LIN {X 27.783,Y -37.308,Z -57.523,A -90.000,B 90.000,C 0.000} C_DIS
LIN {X 27.828,Y -37.308,Z -57.428,A -90.000,B 90.000,C 0.000} C_DIS
LIN {X 28.026,Y -37.308,Z -57.054,A -90.000,B 90.000,C 0.000} C_DIS
LIN {X 28.266,Y -37.308,Z -56.705,A -90.000,B 90.000,C 0.000} C_DIS
LIN {X 28.546,Y -37.308,Z -56.387,A -90.000,B 90.000,C 0.000} C_DIS
LIN {X 28.652,Y -37.308,Z -56.277,A -90.000,B 90.000,C 0.000} C_DIS
LIN {X 28.954,Y -37.308,Z -56.010,A -90.000,B 90.000,C 0.000} C_DIS
LIN {X 29.286,Y -37.308,Z -55.783,A -90.000,B 90.000,C 0.000} C_DIS
LIN {X 29.386,Y -37.308,Z -55.729,A -90.000,B 90.000,C 0.000} C_DIS
LIN {X 29.854,Y -37.308,Z -55.488,A -90.000,B 90.000,C 0.000} C_DIS
LIN {X 30.232,Y -37.308,Z -55.349,A -90.000,B 90.000,C 0.000} C_DIS
LIN {X 30.624,Y -37.308,Z -55.258,A -90.000,B 90.000,C 0.000} C_DIS
LIN {X 30.794,Y -37.308,Z -55.228,A -90.000,B 90.000,C 0.000} C_DIS
LIN {X 30.962,Y -37.308,Z -55.200,A -90.000,B 90.000,C 0.000} C_DIS
LIN {X 31.362,Y -37.308,Z -55.158,A -90.000,B 90.000,C 0.000} C_DIS
LIN {X 31.411,Y -37.308,Z -55.158,A -90.000,B 90.000,C 0.000} C_DIS
LIN {X 31.494,Y -37.308,Z -54.811,A -90.000,B 90.000,C 0.000} C_DIS
LIN {X 31.553,Y -37.308,Z -54.530,A -90.000,B 90.000,C 0.000} C_DIS
LIN {X 31.658,Y -37.308,Z -54.086,A -90.000,B 90.000,C 0.000} C_DIS
LIN {X 31.702,Y -37.308,Z -53.930,A -90.000,B 90.000,C 0.000} C_DIS
LIN {X 31.754,Y -37.308,Z -53.727,A -90.000,B 90.000,C 0.000} C_DIS
LIN {X 31.943,Y -37.308,Z -53.228,A -90.000,B 90.000,C 0.000} C_DIS
LIN {X 32.172,Y -37.308,Z -52.712,A -90.000,B 90.000,C 0.000} C_DIS
LIN {X 32.257,Y -37.308,Z -52.537,A -90.000,B 90.000,C 0.000} C_DIS
LIN {X 32.455,Y -37.308,Z -52.163,A -90.000,B 90.000,C 0.000} C_DIS
LIN {X 32.688,Y -37.308,Z -51.810,A -90.000,B 90.000,C 0.000} C_DIS
LIN {X 32.928,Y -37.308,Z -51.461,A -90.000,B 90.000,C 0.000} C_DIS
LIN {X 33.080,Y -37.308,Z -51.265,A -90.000,B 90.000,C 0.000} C_DIS
LIN {X 33.360,Y -37.308,Z -50.947,A -90.000,B 90.000,C 0.000} C_DIS
LIN {X 33.675,Y -37.308,Z -50.664,A -90.000,B 90.000,C 0.000} C_DIS
LIN {X 33.699,Y -37.308,Z -50.645,A -90.000,B 90.000,C 0.000} C_DIS
LIN {X 33.882,Y -37.308,Z -50.469,A -90.000,B 90.000,C 0.000} C_DIS
LIN {X 34.204,Y -37.308,Z -50.181,A -90.000,B 90.000,C 0.000} C_DIS
LIN {X 34.543,Y -37.308,Z -49.942,A -90.000,B 90.000,C 0.000} C_DIS
LIN {X 34.924,Y -37.308,Z -49.737,A -90.000,B 90.000,C 0.000} C_DIS
LIN {X 35.239,Y -37.308,Z -49.567,A -90.000,B 90.000,C 0.000} C_DIS
LIN {X 35.593,Y -37.308,Z -49.385,A -90.000,B 90.000,C 0.000} C_DIS
LIN {X 35.987,Y -37.308,Z -49.230,A -90.000,B 90.000,C 0.000} C_DIS
LIN {X 36.396,Y -37.308,Z -49.121,A -90.000,B 90.000,C 0.000} C_DIS
LIN {X 36.614,Y -37.308,Z -49.080,A -90.000,B 90.000,C 0.000} C_DIS
LIN {X 37.252,Y -37.308,Z -48.939,A -90.000,B 90.000,C 0.000} C_DIS
LIN {X 37.671,Y -37.308,Z -48.880,A -90.000,B 90.000,C 0.000} C_DIS
LIN {X 38.095,Y -37.308,Z -48.870,A -90.000,B 90.000,C 0.000} C_DIS
LIN {X 38.607,Y -37.308,Z -48.891,A -90.000,B 90.000,C 0.000} C_DIS
LIN {X 39.150,Y -37.308,Z -48.910,A -90.000,B 90.000,C 0.000} C_DIS
LIN {X 39.644,Y -37.308,Z -48.933,A -90.000,B 90.000,C 0.000} C_DIS
LIN {X 40.080,Y -37.308,Z -49.001,A -90.000,B 90.000,C 0.000} C_DIS
LIN {X 40.577,Y -37.308,Z -49.119,A -90.000,B 90.000,C 0.000} C_DIS
LIN {X 41.623,Y -37.308,Z -49.377,A -90.000,B 90.000,C 0.000} C_DIS
LIN {X 41.811,Y -37.308,Z -49.428,A -90.000,B 90.000,C 0.000} C_DIS
LIN {X 42.485,Y -37.308,Z -49.639,A -90.000,B 90.000,C 0.000} C_DIS
LIN {X 43.044,Y -37.308,Z -49.852,A -90.000,B 90.000,C 0.000} C_DIS
LIN {X 43.197,Y -37.308,Z -49.901,A -90.000,B 90.000,C 0.000} C_DIS
LIN {X 44.006,Y -37.308,Z -50.170,A -90.000,B 90.000,C 0.000} C_DIS
LIN {X 44.597,Y -37.308,Z -50.272,A -90.000,B 90.000,C 0.000} C_DIS
LIN {X 45.346,Y -37.308,Z -50.195,A -90.000,B 90.000,C 0.000} C_DIS
LIN {X 45.719,Y -37.308,Z -50.136,A -90.000,B 90.000,C 0.000} C_DIS
LIN {X 46.852,Y -37.308,Z -49.935,A -90.000,B 90.000,C 0.000} C_DIS
LIN {X 47.253,Y -37.308,Z -49.893,A -90.000,B 90.000,C 0.000} C_DIS
LIN {X 47.873,Y -37.308,Z -49.867,A -90.000,B 90.000,C 0.000} C_DIS
LIN {X 49.033,Y -37.308,Z -49.780,A -90.000,B 90.000,C 0.000} C_DIS
LIN {X 49.435,Y -37.308,Z -49.789,A -90.000,B 90.000,C 0.000} C_DIS
LIN {X 49.834,Y -37.308,Z -49.846,A -90.000,B 90.000,C 0.000} C_DIS
LIN {X 50.766,Y -37.308,Z -50.075,A -90.000,B 90.000,C 0.000} C_DIS
LIN {X 52.001,Y -37.308,Z -50.317,A -90.000,B 90.000,C 0.000} C_DIS
LIN {X 52.390,Y -37.308,Z -50.424,A -90.000,B 90.000,C 0.000} C_DIS
LIN {X 52.762,Y -37.308,Z -50.578,A -90.000,B 90.000,C 0.000} C_DIS
LIN {X 53.137,Y -37.308,Z -50.764,A -90.000,B 90.000,C 0.000} C_DIS
LIN {X 53.494,Y -37.308,Z -50.992,A -90.000,B 90.000,C 0.000} C_DIS
LIN {X 55.027,Y -37.308,Z -51.985,A -90.000,B 90.000,C 0.000} C_DIS
LIN {X 55.470,Y -37.308,Z -52.261,A -90.000,B 90.000,C 0.000} C_DIS
LIN {X 55.828,Y -37.308,Z -52.489,A -90.000,B 90.000,C 0.000} C_DIS
LIN {X 56.155,Y -37.308,Z -52.757,A -90.000,B 90.000,C 0.000} C_DIS
LIN {X 58.129,Y -37.308,Z -54.502,A -90.000,B 90.000,C 0.000} C_DIS
LIN {X 58.427,Y -37.308,Z -54.756,A -90.000,B 90.000,C 0.000} C_DIS
LIN {X 59.623,Y -37.308,Z -55.989,A -90.000,B 90.000,C 0.000} C_DIS
LIN {X 60.678,Y -37.308,Z -57.127,A -90.000,B 90.000,C 0.000} C_DIS
LIN {X 60.841,Y -37.308,Z -57.318,A -90.000,B 90.000,C 0.000} C_DIS
LIN {X 61.095,Y -37.308,Z -57.631,A -90.000,B 90.000,C 0.000} C_DIS
LIN {X 62.907,Y -37.308,Z -59.964,A -90.000,B 90.000,C 0.000} C_DIS
LIN {X 64.082,Y -37.308,Z -61.532,A -90.000,B 90.000,C 0.000} C_DIS
LIN {X 64.569,Y -37.308,Z -62.202,A -90.000,B 90.000,C 0.000} C_DIS
LIN {X 64.776,Y -37.308,Z -62.508,A -90.000,B 90.000,C 0.000} C_DIS
LIN {X 64.823,Y -37.308,Z -62.584,A -90.000,B 90.000,C 0.000} C_DIS
LIN {X 66.473,Y -37.308,Z -65.119,A -90.000,B 90.000,C 0.000} C_DIS
LIN {X 68.094,Y -37.308,Z -67.394,A -90.000,B 90.000,C 0.000} C_DIS
LIN {X 68.483,Y -37.308,Z -67.868,A -90.000,B 90.000,C 0.000} C_DIS
LIN {X 69.055,Y -37.308,Z -68.557,A -90.000,B 90.000,C 0.000} C_DIS
LIN {X 71.014,Y -37.308,Z -70.453,A -90.000,B 90.000,C 0.000} C_DIS
LIN {X 71.187,Y -37.308,Z -70.608,A -90.000,B 90.000,C 0.000} C_DIS
LIN {X 72.017,Y -37.308,Z -71.360,A -90.000,B 90.000,C 0.000} C_DIS
LIN {X 72.363,Y -37.308,Z -71.676,A -90.000,B 90.000,C 0.000} C_DIS
LIN {X 72.612,Y -37.308,Z -71.901,A -90.000,B 90.000,C 0.000} C_DIS
LIN {X 73.661,Y -37.308,Z -72.861,A -90.000,B 90.000,C 0.000} C_DIS
LIN {X 73.970,Y -37.308,Z -73.159,A -90.000,B 90.000,C 0.000} C_DIS
LIN {X 74.840,Y -37.308,Z -74.023,A -90.000,B 90.000,C 0.000} C_DIS
LIN {X 75.190,Y -37.308,Z -74.381,A -90.000,B 90.000,C 0.000} C_DIS
LIN {X 76.260,Y -37.308,Z -75.552,A -90.000,B 90.000,C 0.000} C_DIS
LIN {X 76.316,Y -37.308,Z -75.610,A -90.000,B 90.000,C 0.000} C_DIS
LIN {X 76.816,Y -37.308,Z -76.175,A -90.000,B 90.000,C 0.000} C_DIS
LIN {X 77.048,Y -37.308,Z -76.388,A -90.000,B 90.000,C 0.000} C_DIS
LIN {X 77.183,Y -37.308,Z -76.518,A -90.000,B 90.000,C 0.000} C_DIS
LIN {X 77.358,Y -37.308,Z -76.656,A -90.000,B 90.000,C 0.000} C_DIS
LIN {X 77.467,Y -37.308,Z -76.752,A -90.000,B 90.000,C 0.000} C_DIS
LIN {X 77.895,Y -37.308,Z -76.631,A -90.000,B 90.000,C 0.000} C_DIS
LIN {X 77.919,Y -37.308,Z -76.212,A -90.000,B 90.000,C 0.000} C_DIS
LIN {X 77.968,Y -37.308,Z -75.699,A -90.000,B 90.000,C 0.000} C_DIS
LIN {X 78.002,Y -37.308,Z -75.376,A -90.000,B 90.000,C 0.000} C_DIS
LIN {X 78.021,Y -37.308,Z -75.002,A -90.000,B 90.000,C 0.000} C_DIS
LIN {X 78.090,Y -37.308,Z -74.174,A -90.000,B 90.000,C 0.000} C_DIS
LIN {X 78.188,Y -37.308,Z -73.133,A -90.000,B 90.000,C 0.000} C_DIS
LIN {X 78.240,Y -37.308,Z -72.633,A -90.000,B 90.000,C 0.000} C_DIS
LIN {X 78.304,Y -37.308,Z -72.102,A -90.000,B 90.000,C 0.000} C_DIS
LIN {X 78.457,Y -37.308,Z -71.210,A -90.000,B 90.000,C 0.000} C_DIS
LIN {X 78.569,Y -37.308,Z -70.697,A -90.000,B 90.000,C 0.000} C_DIS
LIN {X 78.787,Y -37.308,Z -69.967,A -90.000,B 90.000,C 0.000} C_DIS
LIN {X 79.031,Y -37.308,Z -69.231,A -90.000,B 90.000,C 0.000} C_DIS
LIN {X 79.184,Y -37.308,Z -68.786,A -90.000,B 90.000,C 0.000} C_DIS
LIN {X 79.235,Y -37.308,Z -68.654,A -90.000,B 90.000,C 0.000} C_DIS
LIN {X 79.791,Y -37.308,Z -67.259,A -90.000,B 90.000,C 0.000} C_DIS
LIN {X 80.485,Y -37.308,Z -65.685,A -90.000,B 90.000,C 0.000} C_DIS
LIN {X 80.643,Y -37.308,Z -65.338,A -90.000,B 90.000,C 0.000} C_DIS
LIN {X 81.438,Y -37.308,Z -63.804,A -90.000,B 90.000,C 0.000} C_DIS
LIN {X 81.684,Y -37.308,Z -63.383,A -90.000,B 90.000,C 0.000} C_DIS
LIN {X 82.705,Y -37.308,Z -61.742,A -90.000,B 90.000,C 0.000} C_DIS
LIN {X 84.243,Y -37.308,Z -59.630,A -90.000,B 90.000,C 0.000} C_DIS
LIN {X 85.732,Y -37.308,Z -57.856,A -90.000,B 90.000,C 0.000} C_DIS
LIN {X 86.059,Y -37.308,Z -57.494,A -90.000,B 90.000,C 0.000} C_DIS
LIN {X 87.795,Y -37.308,Z -55.685,A -90.000,B 90.000,C 0.000} C_DIS
LIN {X 89.917,Y -37.308,Z -53.744,A -90.000,B 90.000,C 0.000} C_DIS
LIN {X 90.161,Y -37.308,Z -53.524,A -90.000,B 90.000,C 0.000} C_DIS
LIN {X 92.393,Y -37.308,Z -51.613,A -90.000,B 90.000,C 0.000} C_DIS
LIN {X 94.367,Y -37.308,Z -49.945,A -90.000,B 90.000,C 0.000} C_DIS
LIN {X 96.070,Y -37.308,Z -48.453,A -90.000,B 90.000,C 0.000} C_DIS
LIN {X 96.257,Y -37.308,Z -48.272,A -90.000,B 90.000,C 0.000} C_DIS
LIN {X 97.648,Y -37.308,Z -46.921,A -90.000,B 90.000,C 0.000} C_DIS
LIN {X 99.081,Y -37.308,Z -45.409,A -90.000,B 90.000,C 0.000} C_DIS
LIN {X 100.101,Y -37.308,Z -44.272,A -90.000,B 90.000,C 0.000} C_DIS
LIN {X 101.207,Y -37.308,Z -43.025,A -90.000,B 90.000,C 0.000} C_DIS
LIN {X 101.612,Y -37.308,Z -42.577,A -90.000,B 90.000,C 0.000} C_DIS
LIN {X 101.626,Y -37.308,Z -42.420,A -90.000,B 90.000,C 0.000} C_DIS
LIN {X 101.691,Y -37.308,Z -42.047,A -90.000,B 90.000,C 0.000} C_DIS
LIN {X 101.806,Y -37.308,Z -41.686,A -90.000,B 90.000,C 0.000} C_DIS
LIN {X 101.994,Y -37.308,Z -41.214,A -90.000,B 90.000,C 0.000} C_DIS
LIN {X 102.025,Y -37.308,Z -41.152,A -90.000,B 90.000,C 0.000} C_DIS
LIN {X 102.202,Y -37.308,Z -40.761,A -90.000,B 90.000,C 0.000} C_DIS
LIN {X 102.385,Y -37.308,Z -40.403,A -90.000,B 90.000,C 0.000} C_DIS
LIN {X 102.612,Y -37.308,Z -40.071,A -90.000,B 90.000,C 0.000} C_DIS
LIN {X 102.730,Y -37.308,Z -39.902,A -90.000,B 90.000,C 0.000} C_DIS
LIN {X 102.912,Y -37.308,Z -39.648,A -90.000,B 90.000,C 0.000} C_DIS
LIN {X 103.192,Y -37.308,Z -39.330,A -90.000,B 90.000,C 0.000} C_DIS
LIN {X 103.547,Y -37.308,Z -38.940,A -90.000,B 90.000,C 0.000} C_DIS
LIN {X 103.822,Y -37.308,Z -38.655,A -90.000,B 90.000,C 0.000} C_DIS
LIN {X 104.164,Y -37.308,Z -38.336,A -90.000,B 90.000,C 0.000} C_DIS
LIN {X 104.977,Y -37.308,Z -37.701,A -90.000,B 90.000,C 0.000} C_DIS
LIN {X 105.078,Y -37.308,Z -37.633,A -90.000,B 90.000,C 0.000} C_DIS
LIN {X 105.655,Y -37.308,Z -37.264,A -90.000,B 90.000,C 0.000} C_DIS
LIN {X 105.940,Y -37.308,Z -37.096,A -90.000,B 90.000,C 0.000} C_DIS
LIN {X 106.153,Y -37.308,Z -36.976,A -90.000,B 90.000,C 0.000} C_DIS
LIN {X 106.829,Y -37.308,Z -36.620,A -90.000,B 90.000,C 0.000} C_DIS
LIN {X 107.319,Y -37.308,Z -36.397,A -90.000,B 90.000,C 0.000} C_DIS
LIN {X 107.789,Y -37.308,Z -36.194,A -90.000,B 90.000,C 0.000} C_DIS
LIN {X 108.086,Y -37.308,Z -36.090,A -90.000,B 90.000,C 0.000} C_DIS
LIN {X 108.258,Y -37.308,Z -36.019,A -90.000,B 90.000,C 0.000} C_DIS
LIN {X 108.979,Y -37.308,Z -35.792,A -90.000,B 90.000,C 0.000} C_DIS
LIN {X 109.140,Y -37.308,Z -35.743,A -90.000,B 90.000,C 0.000} C_DIS
LIN {X 109.144,Y -37.308,Z -35.743,A -90.000,B 90.000,C 0.000} C_DIS
LIN {X 109.388,Y -37.308,Z -35.695,A -90.000,B 90.000,C 0.000} C_DIS
LIN {X 109.502,Y -37.308,Z -35.667,A -90.000,B 90.000,C 0.000} C_DIS
LIN {X 109.960,Y -37.308,Z -35.576,A -90.000,B 90.000,C 0.000} C_DIS
LIN {X 110.091,Y -37.308,Z -35.561,A -90.000,B 90.000,C 0.000} C_DIS
LIN {X 110.406,Y -37.308,Z -35.533,A -90.000,B 90.000,C 0.000} C_DIS
LIN {X 111.018,Y -37.308,Z -35.499,A -90.000,B 90.000,C 0.000} C_DIS
LIN {X 111.215,Y -37.308,Z -35.502,A -90.000,B 90.000,C 0.000} C_DIS
LIN {X 111.681,Y -37.308,Z -35.527,A -90.000,B 90.000,C 0.000} C_DIS
LIN {X 111.909,Y -37.308,Z -35.558,A -90.000,B 90.000,C 0.000} C_DIS
LIN {X 112.477,Y -37.308,Z -35.646,A -90.000,B 90.000,C 0.000} C_DIS
LIN {X 112.566,Y -37.308,Z -35.662,A -90.000,B 90.000,C 0.000} C_DIS
LIN {X 112.925,Y -37.308,Z -35.754,A -90.000,B 90.000,C 0.000} C_DIS
LIN {X 113.204,Y -37.308,Z -35.833,A -90.000,B 90.000,C 0.000} C_DIS
LIN {X 113.356,Y -37.308,Z -35.884,A -90.000,B 90.000,C 0.000} C_DIS
LIN {X 113.804,Y -37.308,Z -36.063,A -90.000,B 90.000,C 0.000} C_DIS
LIN {X 114.126,Y -37.308,Z -36.203,A -90.000,B 90.000,C 0.000} C_DIS
LIN {X 114.559,Y -37.308,Z -36.430,A -90.000,B 90.000,C 0.000} C_DIS
LIN {X 114.670,Y -37.308,Z -36.491,A -90.000,B 90.000,C 0.000} C_DIS
LIN {X 115.072,Y -37.308,Z -36.761,A -90.000,B 90.000,C 0.000} C_DIS
LIN {X 115.167,Y -37.308,Z -36.826,A -90.000,B 90.000,C 0.000} C_DIS
LIN {X 115.539,Y -37.308,Z -37.137,A -90.000,B 90.000,C 0.000} C_DIS
LIN {X 115.917,Y -37.308,Z -37.524,A -90.000,B 90.000,C 0.000} C_DIS
LIN {X 116.146,Y -37.308,Z -37.789,A -90.000,B 90.000,C 0.000} C_DIS
LIN {X 116.447,Y -37.308,Z -38.171,A -90.000,B 90.000,C 0.000} C_DIS
LIN {X 116.712,Y -37.308,Z -38.589,A -90.000,B 90.000,C 0.000} C_DIS
LIN {X 116.932,Y -37.308,Z -39.033,A -90.000,B 90.000,C 0.000} C_DIS
LIN {X 117.068,Y -37.308,Z -39.374,A -90.000,B 90.000,C 0.000} C_DIS
LIN {X 117.239,Y -37.308,Z -39.829,A -90.000,B 90.000,C 0.000} C_DIS
LIN {X 117.363,Y -37.308,Z -40.300,A -90.000,B 90.000,C 0.000} C_DIS
LIN {X 117.418,Y -37.308,Z -40.556,A -90.000,B 90.000,C 0.000} C_DIS
LIN {X 117.434,Y -37.308,Z -40.652,A -90.000,B 90.000,C 0.000} C_DIS
LIN {X 117.445,Y -37.308,Z -40.703,A -90.000,B 90.000,C 0.000} C_DIS
LIN {X 117.520,Y -37.308,Z -41.184,A -90.000,B 90.000,C 0.000} C_DIS
LIN {X 117.534,Y -37.308,Z -41.338,A -90.000,B 90.000,C 0.000} C_DIS
LIN {X 117.557,Y -37.308,Z -41.494,A -90.000,B 90.000,C 0.000} C_DIS
LIN {X 117.568,Y -37.308,Z -41.588,A -90.000,B 90.000,C 0.000} C_DIS
LIN {X 117.593,Y -37.308,Z -41.888,A -90.000,B 90.000,C 0.000} C_DIS
LIN {X 117.621,Y -37.308,Z -42.441,A -90.000,B 90.000,C 0.000} C_DIS
LIN {X 117.621,Y -37.308,Z -42.504,A -90.000,B 90.000,C 0.000} C_DIS
LIN {X 117.609,Y -37.308,Z -42.823,A -90.000,B 90.000,C 0.000} C_DIS
LIN {X 117.574,Y -37.308,Z -43.327,A -90.000,B 90.000,C 0.000} C_DIS
LIN {X 117.535,Y -37.308,Z -43.597,A -90.000,B 90.000,C 0.000} C_DIS
LIN {X 117.515,Y -37.308,Z -43.765,A -90.000,B 90.000,C 0.000} C_DIS
LIN {X 117.420,Y -37.308,Z -44.327,A -90.000,B 90.000,C 0.000} C_DIS
LIN {X 117.355,Y -37.308,Z -44.632,A -90.000,B 90.000,C 0.000} C_DIS
LIN {X 117.213,Y -37.308,Z -45.246,A -90.000,B 90.000,C 0.000} C_DIS
LIN {X 117.018,Y -37.308,Z -45.907,A -90.000,B 90.000,C 0.000} C_DIS
LIN {X 116.919,Y -37.308,Z -46.197,A -90.000,B 90.000,C 0.000} C_DIS
LIN {X 116.801,Y -37.308,Z -46.518,A -90.000,B 90.000,C 0.000} C_DIS
LIN {X 116.580,Y -37.308,Z -47.122,A -90.000,B 90.000,C 0.000} C_DIS
LIN {X 116.189,Y -37.308,Z -48.024,A -90.000,B 90.000,C 0.000} C_DIS
LIN {X 116.163,Y -37.308,Z -48.081,A -90.000,B 90.000,C 0.000} C_DIS
LIN {X 115.979,Y -37.308,Z -48.453,A -90.000,B 90.000,C 0.000} C_DIS
LIN {X 115.416,Y -37.308,Z -49.575,A -90.000,B 90.000,C 0.000} C_DIS
LIN {X 114.891,Y -37.308,Z -50.587,A -90.000,B 90.000,C 0.000} C_DIS
LIN {X 114.226,Y -37.308,Z -51.881,A -90.000,B 90.000,C 0.000} C_DIS
LIN {X 113.568,Y -37.308,Z -53.216,A -90.000,B 90.000,C 0.000} C_DIS
LIN {X 113.065,Y -37.308,Z -54.322,A -90.000,B 90.000,C 0.000} C_DIS
LIN {X 112.409,Y -37.308,Z -55.890,A -90.000,B 90.000,C 0.000} C_DIS
LIN {X 111.769,Y -37.308,Z -57.560,A -90.000,B 90.000,C 0.000} C_DIS
LIN {X 111.219,Y -37.308,Z -59.116,A -90.000,B 90.000,C 0.000} C_DIS
LIN {X 110.657,Y -37.308,Z -60.831,A -90.000,B 90.000,C 0.000} C_DIS
LIN {X 109.992,Y -37.308,Z -62.895,A -90.000,B 90.000,C 0.000} C_DIS
LIN {X 109.781,Y -37.308,Z -63.530,A -90.000,B 90.000,C 0.000} C_DIS
LIN {X 109.259,Y -37.308,Z -65.073,A -90.000,B 90.000,C 0.000} C_DIS
LIN {X 108.355,Y -37.308,Z -67.559,A -90.000,B 90.000,C 0.000} C_DIS
LIN {X 108.258,Y -37.308,Z -67.822,A -90.000,B 90.000,C 0.000} C_DIS
LIN {X 107.712,Y -37.308,Z -69.200,A -90.000,B 90.000,C 0.000} C_DIS
LIN {X 107.296,Y -37.308,Z -70.239,A -90.000,B 90.000,C 0.000} C_DIS
LIN {X 106.241,Y -37.308,Z -72.695,A -90.000,B 90.000,C 0.000} C_DIS
LIN {X 105.408,Y -37.308,Z -74.448,A -90.000,B 90.000,C 0.000} C_DIS
LIN {X 105.152,Y -37.308,Z -74.992,A -90.000,B 90.000,C 0.000} C_DIS
LIN {X 104.942,Y -37.308,Z -75.419,A -90.000,B 90.000,C 0.000} C_DIS
LIN {X 104.350,Y -37.308,Z -76.554,A -90.000,B 90.000,C 0.000} C_DIS
LIN {X 103.829,Y -37.308,Z -77.561,A -90.000,B 90.000,C 0.000} C_DIS
LIN {X 103.505,Y -37.308,Z -78.115,A -90.000,B 90.000,C 0.000} C_DIS
LIN {X 102.739,Y -37.308,Z -79.438,A -90.000,B 90.000,C 0.000} C_DIS
LIN {X 102.687,Y -37.308,Z -79.522,A -90.000,B 90.000,C 0.000} C_DIS
LIN {X 102.486,Y -37.308,Z -79.842,A -90.000,B 90.000,C 0.000} C_DIS
LIN {X 102.202,Y -37.308,Z -80.282,A -90.000,B 90.000,C 0.000} C_DIS
LIN {X 101.601,Y -37.308,Z -81.177,A -90.000,B 90.000,C 0.000} C_DIS
LIN {X 101.413,Y -37.308,Z -81.461,A -90.000,B 90.000,C 0.000} C_DIS
LIN {X 100.818,Y -37.308,Z -82.283,A -90.000,B 90.000,C 0.000} C_DIS
LIN {X 100.396,Y -37.308,Z -82.874,A -90.000,B 90.000,C 0.000} C_DIS
LIN {X 100.080,Y -37.308,Z -83.291,A -90.000,B 90.000,C 0.000} C_DIS
LIN {X 99.391,Y -37.308,Z -84.212,A -90.000,B 90.000,C 0.000} C_DIS
LIN {X 99.199,Y -37.308,Z -84.466,A -90.000,B 90.000,C 0.000} C_DIS
LIN {X 98.501,Y -37.308,Z -85.360,A -90.000,B 90.000,C 0.000} C_DIS
LIN {X 97.955,Y -37.308,Z -86.052,A -90.000,B 90.000,C 0.000} C_DIS
LIN {X 97.697,Y -37.308,Z -86.353,A -90.000,B 90.000,C 0.000} C_DIS
LIN {X 97.117,Y -37.308,Z -87.019,A -90.000,B 90.000,C 0.000} C_DIS
LIN {X 96.168,Y -37.308,Z -88.096,A -90.000,B 90.000,C 0.000} C_DIS
LIN {X 95.830,Y -37.308,Z -88.489,A -90.000,B 90.000,C 0.000} C_DIS
LIN {X 95.669,Y -37.308,Z -88.713,A -90.000,B 90.000,C 0.000} C_DIS
LIN {X 95.534,Y -37.308,Z -88.984,A -90.000,B 90.000,C 0.000} C_DIS
LIN {X 95.329,Y -37.308,Z -89.612,A -90.000,B 90.000,C 0.000} C_DIS
LIN {X 95.189,Y -37.308,Z -90.309,A -90.000,B 90.000,C 0.000} C_DIS
LIN {X 95.136,Y -37.308,Z -90.566,A -90.000,B 90.000,C 0.000} C_DIS
LIN {X 95.054,Y -37.308,Z -90.923,A -90.000,B 90.000,C 0.000} C_DIS
LIN {X 94.803,Y -37.308,Z -92.319,A -90.000,B 90.000,C 0.000} C_DIS
LIN {X 94.762,Y -37.308,Z -92.589,A -90.000,B 90.000,C 0.000} C_DIS
LIN {X 94.634,Y -37.308,Z -93.349,A -90.000,B 90.000,C 0.000} C_DIS
LIN {X 94.489,Y -37.308,Z -94.384,A -90.000,B 90.000,C 0.000} C_DIS
LIN {X 94.420,Y -37.308,Z -94.758,A -90.000,B 90.000,C 0.000} C_DIS
LIN {X 94.228,Y -37.308,Z -95.949,A -90.000,B 90.000,C 0.000} C_DIS
LIN {X 94.143,Y -37.308,Z -96.364,A -90.000,B 90.000,C 0.000} C_DIS
LIN {X 94.122,Y -37.308,Z -96.442,A -90.000,B 90.000,C 0.000} C_DIS
LIN {X 94.033,Y -37.308,Z -96.801,A -90.000,B 90.000,C 0.000} C_DIS
LIN {X 93.828,Y -37.308,Z -97.522,A -90.000,B 90.000,C 0.000} C_DIS
LIN {X 93.705,Y -37.308,Z -97.887,A -90.000,B 90.000,C 0.000} C_DIS
LIN {X 93.464,Y -37.308,Z -98.466,A -90.000,B 90.000,C 0.000} C_DIS
LIN {X 93.348,Y -37.308,Z -98.754,A -90.000,B 90.000,C 0.000} C_DIS
LIN {X 93.168,Y -37.308,Z -99.137,A -90.000,B 90.000,C 0.000} C_DIS
LIN {X 92.654,Y -37.308,Z -100.134,A -90.000,B 90.000,C 0.000} C_DIS
LIN {X 92.349,Y -37.308,Z -100.712,A -90.000,B 90.000,C 0.000} C_DIS
LIN {X 92.295,Y -37.308,Z -100.802,A -90.000,B 90.000,C 0.000} C_DIS
LIN {X 92.027,Y -37.308,Z -101.353,A -90.000,B 90.000,C 0.000} C_DIS
LIN {X 91.868,Y -37.308,Z -101.644,A -90.000,B 90.000,C 0.000} C_DIS
LIN {X 91.398,Y -37.308,Z -102.662,A -90.000,B 90.000,C 0.000} C_DIS
LIN {X 91.193,Y -37.308,Z -103.246,A -90.000,B 90.000,C 0.000} C_DIS
LIN {X 91.077,Y -37.308,Z -103.567,A -90.000,B 90.000,C 0.000} C_DIS
LIN {X 90.948,Y -37.308,Z -104.217,A -90.000,B 90.000,C 0.000} C_DIS
LIN {X 90.963,Y -37.308,Z -104.672,A -90.000,B 90.000,C 0.000} C_DIS
LIN {X 91.130,Y -37.308,Z -105.640,A -90.000,B 90.000,C 0.000} C_DIS
LIN {X 91.352,Y -37.308,Z -106.809,A -90.000,B 90.000,C 0.000} C_DIS
LIN {X 91.372,Y -37.308,Z -106.973,A -90.000,B 90.000,C 0.000} C_DIS
LIN {X 91.513,Y -37.308,Z -108.226,A -90.000,B 90.000,C 0.000} C_DIS
LIN {X 91.538,Y -37.308,Z -108.628,A -90.000,B 90.000,C 0.000} C_DIS
LIN {X 91.528,Y -37.308,Z -110.330,A -90.000,B 90.000,C 0.000} C_DIS
LIN {X 91.529,Y -37.308,Z -110.418,A -90.000,B 90.000,C 0.000} C_DIS
LIN {X 91.518,Y -37.308,Z -110.678,A -90.000,B 90.000,C 0.000} C_DIS
LIN {X 91.467,Y -37.308,Z -111.588,A -90.000,B 90.000,C 0.000} C_DIS
LIN {X 91.391,Y -37.308,Z -112.734,A -90.000,B 90.000,C 0.000} C_DIS
LIN {X 91.221,Y -37.308,Z -114.928,A -90.000,B 90.000,C 0.000} C_DIS
LIN {X 91.195,Y -37.308,Z -115.378,A -90.000,B 90.000,C 0.000} C_DIS
LIN {X 91.065,Y -37.308,Z -117.019,A -90.000,B 90.000,C 0.000} C_DIS
LIN {X 91.031,Y -37.308,Z -119.075,A -90.000,B 90.000,C 0.000} C_DIS
LIN {X 91.058,Y -37.308,Z -120.513,A -90.000,B 90.000,C 0.000} C_DIS
LIN {X 91.068,Y -37.308,Z -121.157,A -90.000,B 90.000,C 0.000} C_DIS
LIN {X 91.114,Y -37.308,Z -123.111,A -90.000,B 90.000,C 0.000} C_DIS
LIN {X 91.119,Y -37.308,Z -123.202,A -90.000,B 90.000,C 0.000} C_DIS
LIN {X 91.119,Y -37.308,Z -124.934,A -90.000,B 90.000,C 0.000} C_DIS
LIN {X 91.129,Y -37.308,Z -125.201,A -90.000,B 90.000,C 0.000} C_DIS
LIN {X 91.113,Y -37.308,Z -125.748,A -90.000,B 90.000,C 0.000} C_DIS
LIN {X 91.105,Y -37.308,Z -125.932,A -90.000,B 90.000,C 0.000} C_DIS
LIN {X 91.025,Y -37.308,Z -127.391,A -90.000,B 90.000,C 0.000} C_DIS
LIN {X 90.980,Y -37.308,Z -127.987,A -90.000,B 90.000,C 0.000} C_DIS
LIN {X 90.776,Y -37.308,Z -130.194,A -90.000,B 90.000,C 0.000} C_DIS
LIN {X 90.617,Y -37.308,Z -131.697,A -90.000,B 90.000,C 0.000} C_DIS
LIN {X 90.527,Y -37.308,Z -132.671,A -90.000,B 90.000,C 0.000} C_DIS
LIN {X 90.360,Y -37.308,Z -134.321,A -90.000,B 90.000,C 0.000} C_DIS
LIN {X 90.201,Y -37.308,Z -136.205,A -90.000,B 90.000,C 0.000} C_DIS
LIN {X 90.106,Y -37.308,Z -137.435,A -90.000,B 90.000,C 0.000} C_DIS
LIN {X 89.927,Y -37.308,Z -139.578,A -90.000,B 90.000,C 0.000} C_DIS
LIN {X 89.826,Y -37.308,Z -140.909,A -90.000,B 90.000,C 0.000} C_DIS
LIN {X 89.603,Y -37.308,Z -143.291,A -90.000,B 90.000,C 0.000} C_DIS
LIN {X 89.490,Y -37.308,Z -144.612,A -90.000,B 90.000,C 0.000} C_DIS
LIN {X 89.200,Y -37.308,Z -147.188,A -90.000,B 90.000,C 0.000} C_DIS
LIN {X 89.072,Y -37.308,Z -148.409,A -90.000,B 90.000,C 0.000} C_DIS
LIN {X 88.927,Y -37.308,Z -149.498,A -90.000,B 90.000,C 0.000} C_DIS
LIN {X 88.530,Y -37.308,Z -152.263,A -90.000,B 90.000,C 0.000} C_DIS
LIN {X 88.488,Y -37.308,Z -152.538,A -90.000,B 90.000,C 0.000} C_DIS
LIN {X 88.331,Y -37.308,Z -153.489,A -90.000,B 90.000,C 0.000} C_DIS
LIN {X 87.849,Y -37.308,Z -156.245,A -90.000,B 90.000,C 0.000} C_DIS
LIN {X 87.681,Y -37.308,Z -157.086,A -90.000,B 90.000,C 0.000} C_DIS
LIN {X 87.094,Y -37.308,Z -159.902,A -90.000,B 90.000,C 0.000} C_DIS
LIN {X 86.909,Y -37.308,Z -160.686,A -90.000,B 90.000,C 0.000} C_DIS
LIN {X 86.221,Y -37.308,Z -163.510,A -90.000,B 90.000,C 0.000} C_DIS
LIN {X 85.723,Y -37.308,Z -165.313,A -90.000,B 90.000,C 0.000} C_DIS
LIN {X 85.113,Y -37.308,Z -167.492,A -90.000,B 90.000,C 0.000} C_DIS
LIN {X 84.676,Y -37.308,Z -168.939,A -90.000,B 90.000,C 0.000} C_DIS
LIN {X 84.065,Y -37.308,Z -170.944,A -90.000,B 90.000,C 0.000} C_DIS
LIN {X 83.587,Y -37.308,Z -172.461,A -90.000,B 90.000,C 0.000} C_DIS
LIN {X 83.017,Y -37.308,Z -174.255,A -90.000,B 90.000,C 0.000} C_DIS
LIN {X 82.540,Y -37.308,Z -175.781,A -90.000,B 90.000,C 0.000} C_DIS
LIN {X 82.026,Y -37.308,Z -177.391,A -90.000,B 90.000,C 0.000} C_DIS
LIN {X 81.570,Y -37.308,Z -178.879,A -90.000,B 90.000,C 0.000} C_DIS
LIN {X 81.147,Y -37.308,Z -180.323,A -90.000,B 90.000,C 0.000} C_DIS
LIN {X 80.709,Y -37.308,Z -181.794,A -90.000,B 90.000,C 0.000} C_DIS
LIN {X 80.349,Y -37.308,Z -183.087,A -90.000,B 90.000,C 0.000} C_DIS
LIN {X 79.901,Y -37.308,Z -184.606,A -90.000,B 90.000,C 0.000} C_DIS
LIN {X 79.599,Y -37.308,Z -185.715,A -90.000,B 90.000,C 0.000} C_DIS
LIN {X 79.124,Y -37.308,Z -187.315,A -90.000,B 90.000,C 0.000} C_DIS
LIN {X 78.869,Y -37.308,Z -188.241,A -90.000,B 90.000,C 0.000} C_DIS
LIN {X 78.356,Y -37.308,Z -189.928,A -90.000,B 90.000,C 0.000} C_DIS
LIN {X 78.136,Y -37.308,Z -190.700,A -90.000,B 90.000,C 0.000} C_DIS
LIN {X 77.535,Y -37.308,Z -192.575,A -90.000,B 90.000,C 0.000} C_DIS
LIN {X 77.324,Y -37.308,Z -193.266,A -90.000,B 90.000,C 0.000} C_DIS
LIN {X 76.579,Y -37.308,Z -195.452,A -90.000,B 90.000,C 0.000} C_DIS
LIN {X 76.361,Y -37.308,Z -196.112,A -90.000,B 90.000,C 0.000} C_DIS
LIN {X 75.409,Y -37.308,Z -198.746,A -90.000,B 90.000,C 0.000} C_DIS
LIN {X 75.152,Y -37.308,Z -199.466,A -90.000,B 90.000,C 0.000} C_DIS
LIN {X 74.103,Y -37.308,Z -202.233,A -90.000,B 90.000,C 0.000} C_DIS
LIN {X 73.601,Y -37.308,Z -203.568,A -90.000,B 90.000,C 0.000} C_DIS
LIN {X 71.852,Y -37.308,Z -207.990,A -90.000,B 90.000,C 0.000} C_DIS
LIN {X 69.873,Y -37.308,Z -212.790,A -90.000,B 90.000,C 0.000} C_DIS
LIN {X 67.700,Y -37.308,Z -217.846,A -90.000,B 90.000,C 0.000} C_DIS
LIN {X 65.367,Y -37.308,Z -223.035,A -90.000,B 90.000,C 0.000} C_DIS
LIN {X 65.024,Y -37.308,Z -223.760,A -90.000,B 90.000,C 0.000} C_DIS
LIN {X 64.784,Y -37.308,Z -224.263,A -90.000,B 90.000,C 0.000} C_DIS
LIN {X 62.789,Y -37.308,Z -228.504,A -90.000,B 90.000,C 0.000} C_DIS
LIN {X 62.689,Y -37.308,Z -228.712,A -90.000,B 90.000,C 0.000} C_DIS
LIN {X 62.424,Y -37.308,Z -229.232,A -90.000,B 90.000,C 0.000} C_DIS
LIN {X 60.135,Y -37.308,Z -233.876,A -90.000,B 90.000,C 0.000} C_DIS
LIN {X 59.979,Y -37.308,Z -234.165,A -90.000,B 90.000,C 0.000} C_DIS
LIN {X 57.323,Y -37.308,Z -239.304,A -90.000,B 90.000,C 0.000} C_DIS
LIN {X 55.010,Y -37.308,Z -243.561,A -90.000,B 90.000,C 0.000} C_DIS
LIN {X 55.010,Y -60.000,Z -243.561,A -90.000,B 90.000,C 0.000} C_DIS
LIN {X 98.544,Y -60.000,Z -45.976,A -90.000,B 90.000,C 0.000} C_DIS
LIN {X 98.544,Y -35.308,Z -45.976,A -90.000,B 90.000,C 0.000} C_DIS
LIN {X 98.535,Y -35.309,Z -45.952,A -90.000,B 90.000,C 0.000} C_DIS
LIN {X 98.457,Y -35.348,Z -45.492,A -90.000,B 90.000,C 0.000} C_DIS
LIN {X 98.454,Y -35.360,Z -45.413,A -90.000,B 90.000,C 0.000} C_DIS
LIN {X 98.465,Y -35.379,Z -45.295,A -90.000,B 90.000,C 0.000} C_DIS
LIN {X 98.472,Y -35.389,Z -45.233,A -90.000,B 90.000,C 0.000} C_DIS
LIN {X 98.502,Y -35.427,Z -45.036,A -90.000,B 90.000,C 0.000} C_DIS
LIN {X 98.568,Y -35.475,Z -44.785,A -90.000,B 90.000,C 0.000} C_DIS
LIN {X 98.664,Y -35.537,Z -44.484,A -90.000,B 90.000,C 0.000} C_DIS
LIN {X 98.714,Y -35.569,Z -44.341,A -90.000,B 90.000,C 0.000} C_DIS
LIN {X 98.780,Y -35.607,Z -44.171,A -90.000,B 90.000,C 0.000} C_DIS
LIN {X 98.841,Y -35.642,Z -44.021,A -90.000,B 90.000,C 0.000} C_DIS
LIN {X 98.963,Y -35.713,Z -43.735,A -90.000,B 90.000,C 0.000} C_DIS
LIN {X 99.104,Y -35.781,Z -43.450,A -90.000,B 90.000,C 0.000} C_DIS
LIN {X 99.185,Y -35.821,Z -43.291,A -90.000,B 90.000,C 0.000} C_DIS
LIN {X 99.431,Y -35.914,Z -42.866,A -90.000,B 90.000,C 0.000} C_DIS
LIN {X 99.591,Y -35.969,Z -42.608,A -90.000,B 90.000,C 0.000} C_DIS
LIN {X 99.870,Y -36.063,Z -42.173,A -90.000,B 90.000,C 0.000} C_DIS
LIN {X 100.092,Y -36.118,Z -41.863,A -90.000,B 90.000,C 0.000} C_DIS
LIN {X 100.113,Y -36.108,Z -41.788,A -90.000,B 90.000,C 0.000} C_DIS
LIN {X 100.146,Y -36.092,Z -41.681,A -90.000,B 90.000,C 0.000} C_DIS
LIN {X 100.201,Y -36.076,Z -41.536,A -90.000,B 90.000,C 0.000} C_DIS
LIN {X 100.295,Y -36.054,Z -41.296,A -90.000,B 90.000,C 0.000} C_DIS
LIN {X 100.333,Y -36.040,Z -41.215,A -90.000,B 90.000,C 0.000} C_DIS
LIN {X 100.395,Y -36.021,Z -41.093,A -90.000,B 90.000,C 0.000} C_DIS
LIN {X 100.620,Y -35.963,Z -40.665,A -90.000,B 90.000,C 0.000} C_DIS
LIN {X 100.691,Y -35.949,Z -40.539,A -90.000,B 90.000,C 0.000} C_DIS
LIN {X 100.927,Y -35.881,Z -40.180,A -90.000,B 90.000,C 0.000} C_DIS
LIN {X 101.164,Y -35.828,Z -39.839,A -90.000,B 90.000,C 0.000} C_DIS
LIN {X 101.261,Y -35.802,Z -39.720,A -90.000,B 90.000,C 0.000} C_DIS
LIN {X 101.370,Y -35.783,Z -39.597,A -90.000,B 90.000,C 0.000} C_DIS
LIN {X 101.597,Y -35.745,Z -39.348,A -90.000,B 90.000,C 0.000} C_DIS
LIN {X 101.766,Y -35.718,Z -39.165,A -90.000,B 90.000,C 0.000} C_DIS
LIN {X 101.970,Y -35.680,Z -38.969,A -90.000,B 90.000,C 0.000} C_DIS
LIN {X 102.054,Y -35.667,Z -38.892,A -90.000,B 90.000,C 0.000} C_DIS
LIN {X 102.471,Y -35.624,Z -38.520,A -90.000,B 90.000,C 0.000} C_DIS
LIN {X 102.642,Y -35.606,Z -38.375,A -90.000,B 90.000,C 0.000} C_DIS
LIN {X 102.891,Y -35.576,Z -38.181,A -90.000,B 90.000,C 0.000} C_DIS
LIN {X 103.164,Y -35.547,Z -37.974,A -90.000,B 90.000,C 0.000} C_DIS
LIN {X 103.301,Y -35.535,Z -37.877,A -90.000,B 90.000,C 0.000} C_DIS
LIN {X 103.576,Y -35.511,Z -37.686,A -90.000,B 90.000,C 0.000} C_DIS
LIN {X 103.842,Y -35.497,Z -37.511,A -90.000,B 90.000,C 0.000} C_DIS
LIN {X 104.277,Y -35.472,Z -37.243,A -90.000,B 90.000,C 0.000} C_DIS
LIN {X 104.510,Y -35.455,Z -37.112,A -90.000,B 90.000,C 0.000} C_DIS
LIN {X 104.658,Y -35.448,Z -37.031,A -90.000,B 90.000,C 0.000} C_DIS
LIN {X 104.824,Y -35.443,Z -36.940,A -90.000,B 90.000,C 0.000} C_DIS
LIN {X 105.339,Y -35.420,Z -36.686,A -90.000,B 90.000,C 0.000} C_DIS
LIN {X 105.565,Y -35.412,Z -36.580,A -90.000,B 90.000,C 0.000} C_DIS
LIN {X 105.950,Y -35.400,Z -36.408,A -90.000,B 90.000,C 0.000} C_DIS
LIN {X 106.259,Y -35.393,Z -36.270,A -90.000,B 90.000,C 0.000} C_DIS
LIN {X 106.493,Y -35.387,Z -36.170,A -90.000,B 90.000,C 0.000} C_DIS
LIN {X 106.621,Y -35.383,Z -36.119,A -90.000,B 90.000,C 0.000} C_DIS
LIN {X 106.824,Y -35.383,Z -36.028,A -90.000,B 90.000,C 0.000} C_DIS
LIN {X 107.111,Y -35.381,Z -35.905,A -90.000,B 90.000,C 0.000} C_DIS
LIN {X 107.402,Y -35.378,Z -35.791,A -90.000,B 90.000,C 0.000} C_DIS
LIN {X 107.653,Y -35.374,Z -35.701,A -90.000,B 90.000,C 0.000} C_DIS
LIN {X 107.904,Y -35.375,Z -35.612,A -90.000,B 90.000,C 0.000} C_DIS
LIN {X 108.107,Y -35.372,Z -35.542,A -90.000,B 90.000,C 0.000} C_DIS
LIN {X 108.303,Y -35.373,Z -35.476,A -90.000,B 90.000,C 0.000} C_DIS
LIN {X 108.735,Y -35.370,Z -35.353,A -90.000,B 90.000,C 0.000} C_DIS
LIN {X 109.059,Y -35.365,Z -35.277,A -90.000,B 90.000,C 0.000} C_DIS
LIN {X 109.210,Y -35.366,Z -35.243,A -90.000,B 90.000,C 0.000} C_DIS
LIN {X 109.325,Y -35.365,Z -35.226,A -90.000,B 90.000,C 0.000} C_DIS
LIN {X 109.618,Y -35.360,Z -35.182,A -90.000,B 90.000,C 0.000} C_DIS
LIN {X 109.909,Y -35.356,Z -35.146,A -90.000,B 90.000,C 0.000} C_DIS
LIN {X 110.101,Y -35.356,Z -35.122,A -90.000,B 90.000,C 0.000} C_DIS
LIN {X 110.589,Y -35.351,Z -35.113,A -90.000,B 90.000,C 0.000} C_DIS
LIN {X 110.947,Y -35.346,Z -35.118,A -90.000,B 90.000,C 0.000} C_DIS
LIN {X 111.433,Y -35.340,Z -35.159,A -90.000,B 90.000,C 0.000} C_DIS
LIN {X 111.510,Y -35.338,Z -35.172,A -90.000,B 90.000,C 0.000} C_DIS
LIN {X 111.837,Y -35.333,Z -35.233,A -90.000,B 90.000,C 0.000} C_DIS
LIN {X 112.069,Y -35.331,Z -35.277,A -90.000,B 90.000,C 0.000} C_DIS
LIN {X 112.408,Y -35.327,Z -35.363,A -90.000,B 90.000,C 0.000} C_DIS
LIN {X 112.933,Y -35.321,Z -35.521,A -90.000,B 90.000,C 0.000} C_DIS
LIN {X 113.059,Y -35.321,Z -35.562,A -90.000,B 90.000,C 0.000} C_DIS
LIN {X 113.521,Y -35.317,Z -35.754,A -90.000,B 90.000,C 0.000} C_DIS
LIN {X 113.997,Y -35.314,Z -35.982,A -90.000,B 90.000,C 0.000} C_DIS
LIN {X 114.411,Y -35.313,Z -36.206,A -90.000,B 90.000,C 0.000} C_DIS
LIN {X 114.550,Y -35.312,Z -36.292,A -90.000,B 90.000,C 0.000} C_DIS
LIN {X 114.946,Y -35.311,Z -36.562,A -90.000,B 90.000,C 0.000} C_DIS
LIN {X 115.059,Y -35.310,Z -36.652,A -90.000,B 90.000,C 0.000} C_DIS
LIN {X 115.208,Y -35.309,Z -36.777,A -90.000,B 90.000,C 0.000} C_DIS
LIN {X 115.426,Y -35.309,Z -36.960,A -90.000,B 90.000,C 0.000} C_DIS
LIN {X 115.524,Y -35.309,Z -37.050,A -90.000,B 90.000,C 0.000} C_DIS
LIN {X 115.859,Y -35.309,Z -37.397,A -90.000,B 90.000,C 0.000} C_DIS
LIN {X 116.077,Y -35.309,Z -37.628,A -90.000,B 90.000,C 0.000} C_DIS
LIN {X 116.439,Y -35.309,Z -38.088,A -90.000,B 90.000,C 0.000} C_DIS
LIN {X 116.700,Y -35.309,Z -38.500,A -90.000,B 90.000,C 0.000} C_DIS
LIN {X 116.922,Y -35.309,Z -38.948,A -90.000,B 90.000,C 0.000} C_DIS
LIN {X 117.057,Y -35.309,Z -39.246,A -90.000,B 90.000,C 0.000} C_DIS
LIN {X 117.109,Y -35.309,Z -39.378,A -90.000,B 90.000,C 0.000} C_DIS
LIN {X 117.260,Y -35.309,Z -39.781,A -90.000,B 90.000,C 0.000} C_DIS
LIN {X 117.387,Y -35.309,Z -40.266,A -90.000,B 90.000,C 0.000} C_DIS
LIN {X 117.464,Y -35.309,Z -40.606,A -90.000,B 90.000,C 0.000} C_DIS
LIN {X 117.538,Y -35.309,Z -41.090,A -90.000,B 90.000,C 0.000} C_DIS
LIN {X 117.594,Y -35.309,Z -41.507,A -90.000,B 90.000,C 0.000} C_DIS
LIN {X 117.631,Y -35.309,Z -41.891,A -90.000,B 90.000,C 0.000} C_DIS
LIN {X 117.659,Y -35.309,Z -42.462,A -90.000,B 90.000,C 0.000} C_DIS
LIN {X 117.668,Y -35.309,Z -42.690,A -90.000,B 90.000,C 0.000} C_DIS
LIN {X 117.665,Y -35.309,Z -42.838,A -90.000,B 90.000,C 0.000} C_DIS
LIN {X 117.651,Y -35.310,Z -43.213,A -90.000,B 90.000,C 0.000} C_DIS
LIN {X 117.609,Y -35.310,Z -43.701,A -90.000,B 90.000,C 0.000} C_DIS
LIN {X 117.565,Y -35.311,Z -44.130,A -90.000,B 90.000,C 0.000} C_DIS
LIN {X 117.486,Y -35.313,Z -44.650,A -90.000,B 90.000,C 0.000} C_DIS
LIN {X 117.393,Y -35.314,Z -45.141,A -90.000,B 90.000,C 0.000} C_DIS
LIN {X 117.255,Y -35.317,Z -45.755,A -90.000,B 90.000,C 0.000} C_DIS
LIN {X 117.103,Y -35.318,Z -46.266,A -90.000,B 90.000,C 0.000} C_DIS
LIN {X 116.899,Y -35.323,Z -46.941,A -90.000,B 90.000,C 0.000} C_DIS
LIN {X 116.647,Y -35.324,Z -47.594,A -90.000,B 90.000,C 0.000} C_DIS
LIN {X 116.555,Y -35.325,Z -47.833,A -90.000,B 90.000,C 0.000} C_DIS
LIN {X 116.369,Y -35.327,Z -48.284,A -90.000,B 90.000,C 0.000} C_DIS
LIN {X 115.872,Y -35.332,Z -49.352,A -90.000,B 90.000,C 0.000} C_DIS
LIN {X 115.522,Y -35.333,Z -50.050,A -90.000,B 90.000,C 0.000} C_DIS
LIN {X 115.174,Y -35.334,Z -50.733,A -90.000,B 90.000,C 0.000} C_DIS
LIN {X 114.626,Y -35.334,Z -51.801,A -90.000,B 90.000,C 0.000} C_DIS
LIN {X 113.947,Y -35.334,Z -53.171,A -90.000,B 90.000,C 0.000} C_DIS
LIN {X 113.872,Y -35.335,Z -53.334,A -90.000,B 90.000,C 0.000} C_DIS
LIN {X 113.284,Y -35.333,Z -54.612,A -90.000,B 90.000,C 0.000} C_DIS
LIN {X 112.688,Y -35.332,Z -56.010,A -90.000,B 90.000,C 0.000} C_DIS
LIN {X 112.182,Y -35.331,Z -57.325,A -90.000,B 90.000,C 0.000} C_DIS
LIN {X 111.584,Y -35.335,Z -59.067,A -90.000,B 90.000,C 0.000} C_DIS
LIN {X 111.009,Y -35.343,Z -60.948,A -90.000,B 90.000,C 0.000} C_DIS
LIN {X 110.501,Y -35.351,Z -62.658,A -90.000,B 90.000,C 0.000} C_DIS
LIN {X 110.387,Y -35.352,Z -63.027,A -90.000,B 90.000,C 0.000} C_DIS
LIN {X 109.803,Y -35.360,Z -64.869,A -90.000,B 90.000,C 0.000} C_DIS
LIN {X 109.580,Y -35.361,Z -65.520,A -90.000,B 90.000,C 0.000} C_DIS
LIN {X 109.452,Y -35.362,Z -65.890,A -90.000,B 90.000,C 0.000} C_DIS
LIN {X 108.868,Y -35.366,Z -67.540,A -90.000,B 90.000,C 0.000} C_DIS
LIN {X 108.571,Y -35.364,Z -68.305,A -90.000,B 90.000,C 0.000} C_DIS
LIN {X 107.922,Y -35.366,Z -69.959,A -90.000,B 90.000,C 0.000} C_DIS
LIN {X 107.688,Y -35.364,Z -70.516,A -90.000,B 90.000,C 0.000} C_DIS
LIN {X 107.087,Y -35.367,Z -71.942,A -90.000,B 90.000,C 0.000} C_DIS
LIN {X 106.889,Y -35.367,Z -72.406,A -90.000,B 90.000,C 0.000} C_DIS
LIN {X 106.678,Y -35.364,Z -72.870,A -90.000,B 90.000,C 0.000} C_DIS
LIN {X 106.286,Y -35.368,Z -73.728,A -90.000,B 90.000,C 0.000} C_DIS
LIN {X 105.598,Y -35.370,Z -75.197,A -90.000,B 90.000,C 0.000} C_DIS
LIN {X 105.283,Y -35.368,Z -75.816,A -90.000,B 90.000,C 0.000} C_DIS
LIN {X 104.494,Y -35.371,Z -77.356,A -90.000,B 90.000,C 0.000} C_DIS
LIN {X 104.241,Y -35.366,Z -77.802,A -90.000,B 90.000,C 0.000} C_DIS
LIN {X 103.846,Y -35.368,Z -78.492,A -90.000,B 90.000,C 0.000} C_DIS
LIN {X 103.418,Y -35.369,Z -79.240,A -90.000,B 90.000,C 0.000} C_DIS
LIN {X 103.151,Y -35.367,Z -79.688,A -90.000,B 90.000,C 0.000} C_DIS
LIN {X 102.606,Y -35.369,Z -80.554,A -90.000,B 90.000,C 0.000} C_DIS
LIN {X 102.123,Y -35.375,Z -81.317,A -90.000,B 90.000,C 0.000} C_DIS
LIN {X 101.790,Y -35.373,Z -81.798,A -90.000,B 90.000,C 0.000} C_DIS
LIN {X 101.157,Y -35.378,Z -82.711,A -90.000,B 90.000,C 0.000} C_DIS
LIN {X 100.811,Y -35.377,Z -83.189,A -90.000,B 90.000,C 0.000} C_DIS
LIN {X 99.521,Y -35.390,Z -84.973,A -90.000,B 90.000,C 0.000} C_DIS
LIN {X 98.945,Y -35.400,Z -85.765,A -90.000,B 90.000,C 0.000} C_DIS
LIN {X 98.414,Y -35.409,Z -86.479,A -90.000,B 90.000,C 0.000} C_DIS
LIN {X 97.879,Y -35.430,Z -87.193,A -90.000,B 90.000,C 0.000} C_DIS
LIN {X 97.087,Y -35.458,Z -88.201,A -90.000,B 90.000,C 0.000} C_DIS
LIN {X 97.060,Y -35.461,Z -88.242,A -90.000,B 90.000,C 0.000} C_DIS
LIN {X 96.978,Y -35.480,Z -88.404,A -90.000,B 90.000,C 0.000} C_DIS
LIN {X 96.844,Y -35.541,Z -88.745,A -90.000,B 90.000,C 0.000} C_DIS
LIN {X 96.739,Y -35.593,Z -89.008,A -90.000,B 90.000,C 0.000} C_DIS
LIN {X 96.677,Y -35.625,Z -89.160,A -90.000,B 90.000,C 0.000} C_DIS
LIN {X 96.636,Y -35.654,Z -89.291,A -90.000,B 90.000,C 0.000} C_DIS
LIN {X 96.601,Y -35.672,Z -89.422,A -90.000,B 90.000,C 0.000} C_DIS
LIN {X 96.491,Y -35.709,Z -89.916,A -90.000,B 90.000,C 0.000} C_DIS
LIN {X 96.396,Y -35.715,Z -90.447,A -90.000,B 90.000,C 0.000} C_DIS
LIN {X 96.331,Y -35.730,Z -90.853,A -90.000,B 90.000,C 0.000} C_DIS
LIN {X 96.279,Y -35.747,Z -91.174,A -90.000,B 90.000,C 0.000} C_DIS
LIN {X 96.209,Y -35.760,Z -91.656,A -90.000,B 90.000,C 0.000} C_DIS
LIN {X 96.105,Y -35.766,Z -92.270,A -90.000,B 90.000,C 0.000} C_DIS
LIN {X 96.049,Y -35.770,Z -92.621,A -90.000,B 90.000,C 0.000} C_DIS
LIN {X 95.974,Y -35.772,Z -93.103,A -90.000,B 90.000,C 0.000} C_DIS
LIN {X 95.901,Y -35.777,Z -93.572,A -90.000,B 90.000,C 0.000} C_DIS
LIN {X 95.813,Y -35.778,Z -94.213,A -90.000,B 90.000,C 0.000} C_DIS
LIN {X 95.750,Y -35.773,Z -94.616,A -90.000,B 90.000,C 0.000} C_DIS
LIN {X 95.686,Y -35.778,Z -94.999,A -90.000,B 90.000,C 0.000} C_DIS
LIN {X 95.558,Y -35.782,Z -95.817,A -90.000,B 90.000,C 0.000} C_DIS
LIN {X 95.477,Y -35.770,Z -96.222,A -90.000,B 90.000,C 0.000} C_DIS
LIN {X 95.387,Y -35.765,Z -96.629,A -90.000,B 90.000,C 0.000} C_DIS
LIN {X 95.328,Y -35.768,Z -96.876,A -90.000,B 90.000,C 0.000} C_DIS
LIN {X 95.257,Y -35.768,Z -97.160,A -90.000,B 90.000,C 0.000} C_DIS
LIN {X 95.216,Y -35.771,Z -97.315,A -90.000,B 90.000,C 0.000} C_DIS
LIN {X 95.085,Y -35.759,Z -97.731,A -90.000,B 90.000,C 0.000} C_DIS
LIN {X 95.052,Y -35.755,Z -97.828,A -90.000,B 90.000,C 0.000} C_DIS
LIN {X 94.883,Y -35.745,Z -98.297,A -90.000,B 90.000,C 0.000} C_DIS
LIN {X 94.837,Y -35.746,Z -98.418,A -90.000,B 90.000,C 0.000} C_DIS
LIN {X 94.735,Y -35.753,Z -98.685,A -90.000,B 90.000,C 0.000} C_DIS
LIN {X 94.515,Y -35.744,Z -99.193,A -90.000,B 90.000,C 0.000} C_DIS
LIN {X 94.475,Y -35.743,Z -99.284,A -90.000,B 90.000,C 0.000} C_DIS
LIN {X 94.301,Y -35.749,Z -99.670,A -90.000,B 90.000,C 0.000} C_DIS
LIN {X 93.927,Y -35.775,Z -100.467,A -90.000,B 90.000,C 0.000} C_DIS
LIN {X 93.617,Y -35.816,Z -101.160,A -90.000,B 90.000,C 0.000} C_DIS
LIN {X 93.503,Y -35.824,Z -101.394,A -90.000,B 90.000,C 0.000} C_DIS
LIN {X 93.478,Y -35.827,Z -101.442,A -90.000,B 90.000,C 0.000} C_DIS
LIN {X 93.451,Y -35.828,Z -101.500,A -90.000,B 90.000,C 0.000} C_DIS
LIN {X 93.238,Y -35.850,Z -101.987,A -90.000,B 90.000,C 0.000} C_DIS
LIN {X 93.109,Y -35.868,Z -102.266,A -90.000,B 90.000,C 0.000} C_DIS
LIN {X 92.922,Y -35.883,Z -102.707,A -90.000,B 90.000,C 0.000} C_DIS
LIN {X 92.733,Y -35.919,Z -103.202,A -90.000,B 90.000,C 0.000} C_DIS
LIN {X 92.585,Y -35.927,Z -103.648,A -90.000,B 90.000,C 0.000} C_DIS
LIN {X 92.500,Y -35.954,Z -103.960,A -90.000,B 90.000,C 0.000} C_DIS
LIN {X 92.427,Y -35.956,Z -104.339,A -90.000,B 90.000,C 0.000} C_DIS
LIN {X 92.425,Y -35.954,Z -104.358,A -90.000,B 90.000,C 0.000} C_DIS
LIN {X 92.428,Y -35.952,Z -104.523,A -90.000,B 90.000,C 0.000} C_DIS
LIN {X 92.461,Y -35.921,Z -104.879,A -90.000,B 90.000,C 0.000} C_DIS
LIN {X 92.540,Y -35.915,Z -105.374,A -90.000,B 90.000,C 0.000} C_DIS
LIN {X 92.605,Y -35.907,Z -105.761,A -90.000,B 90.000,C 0.000} C_DIS
LIN {X 92.751,Y -35.904,Z -106.544,A -90.000,B 90.000,C 0.000} C_DIS
LIN {X 92.779,Y -35.908,Z -106.717,A -90.000,B 90.000,C 0.000} C_DIS
LIN {X 92.808,Y -35.914,Z -106.910,A -90.000,B 90.000,C 0.000} C_DIS
LIN {X 92.953,Y -35.923,Z -108.137,A -90.000,B 90.000,C 0.000} C_DIS
LIN {X 92.965,Y -35.927,Z -108.266,A -90.000,B 90.000,C 0.000} C_DIS
LIN {X 92.982,Y -35.927,Z -108.538,A -90.000,B 90.000,C 0.000} C_DIS
LIN {X 92.987,Y -35.930,Z -108.703,A -90.000,B 90.000,C 0.000} C_DIS
LIN {X 92.994,Y -35.947,Z -110.370,A -90.000,B 90.000,C 0.000} C_DIS
LIN {X 92.991,Y -35.945,Z -110.479,A -90.000,B 90.000,C 0.000} C_DIS
LIN {X 92.979,Y -35.945,Z -110.756,A -90.000,B 90.000,C 0.000} C_DIS
LIN {X 92.935,Y -35.956,Z -111.721,A -90.000,B 90.000,C 0.000} C_DIS
LIN {X 92.888,Y -35.970,Z -112.607,A -90.000,B 90.000,C 0.000} C_DIS
LIN {X 92.852,Y -35.970,Z -113.108,A -90.000,B 90.000,C 0.000} C_DIS
LIN {X 92.727,Y -35.996,Z -115.029,A -90.000,B 90.000,C 0.000} C_DIS
LIN {X 92.705,Y -35.997,Z -115.423,A -90.000,B 90.000,C 0.000} C_DIS
LIN {X 92.658,Y -36.011,Z -116.164,A -90.000,B 90.000,C 0.000} C_DIS
LIN {X 92.623,Y -36.022,Z -116.741,A -90.000,B 90.000,C 0.000} C_DIS
LIN {X 92.606,Y -36.035,Z -117.092,A -90.000,B 90.000,C 0.000} C_DIS
LIN {X 92.586,Y -36.047,Z -118.921,A -90.000,B 90.000,C 0.000} C_DIS
LIN {X 92.585,Y -36.050,Z -119.074,A -90.000,B 90.000,C 0.000} C_DIS
LIN {X 92.602,Y -36.049,Z -120.011,A -90.000,B 90.000,C 0.000} C_DIS
LIN {X 92.625,Y -36.054,Z -121.125,A -90.000,B 90.000,C 0.000} C_DIS
LIN {X 92.639,Y -36.049,Z -121.876,A -90.000,B 90.000,C 0.000} C_DIS
LIN {X 92.671,Y -36.054,Z -123.052,A -90.000,B 90.000,C 0.000} C_DIS
LIN {X 92.675,Y -36.051,Z -123.190,A -90.000,B 90.000,C 0.000} C_DIS
LIN {X 92.672,Y -36.048,Z -123.853,A -90.000,B 90.000,C 0.000} C_DIS
LIN {X 92.675,Y -36.053,Z -124.903,A -90.000,B 90.000,C 0.000} C_DIS
LIN {X 92.681,Y -36.048,Z -125.139,A -90.000,B 90.000,C 0.000} C_DIS
LIN {X 92.678,Y -36.045,Z -125.283,A -90.000,B 90.000,C 0.000} C_DIS
LIN {X 92.662,Y -36.042,Z -125.752,A -90.000,B 90.000,C 0.000} C_DIS
LIN {X 92.644,Y -36.042,Z -126.147,A -90.000,B 90.000,C 0.000} C_DIS
LIN {X 92.604,Y -36.046,Z -126.917,A -90.000,B 90.000,C 0.000} C_DIS
LIN {X 92.576,Y -36.045,Z -127.416,A -90.000,B 90.000,C 0.000} C_DIS
LIN {X 92.522,Y -36.043,Z -128.129,A -90.000,B 90.000,C 0.000} C_DIS
LIN {X 92.409,Y -36.050,Z -129.421,A -90.000,B 90.000,C 0.000} C_DIS
LIN {X 92.319,Y -36.048,Z -130.365,A -90.000,B 90.000,C 0.000} C_DIS
LIN {X 92.168,Y -36.055,Z -131.852,A -90.000,B 90.000,C 0.000} C_DIS
LIN {X 92.076,Y -36.053,Z -132.828,A -90.000,B 90.000,C 0.000} C_DIS
LIN {X 91.915,Y -36.058,Z -134.466,A -90.000,B 90.000,C 0.000} C_DIS
LIN {X 91.883,Y -36.058,Z -134.842,A -90.000,B 90.000,C 0.000} C_DIS
LIN {X 91.757,Y -36.059,Z -136.331,A -90.000,B 90.000,C 0.000} C_DIS
LIN {X 91.659,Y -36.054,Z -137.565,A -90.000,B 90.000,C 0.000} C_DIS
LIN {X 91.478,Y -36.052,Z -139.702,A -90.000,B 90.000,C 0.000} C_DIS
LIN {X 91.369,Y -36.045,Z -141.053,A -90.000,B 90.000,C 0.000} C_DIS
LIN {X 91.144,Y -36.040,Z -143.429,A -90.000,B 90.000,C 0.000} C_DIS
LIN {X 91.025,Y -36.033,Z -144.743,A -90.000,B 90.000,C 0.000} C_DIS
LIN {X 90.722,Y -36.027,Z -147.395,A -90.000,B 90.000,C 0.000} C_DIS
LIN {X 90.603,Y -36.020,Z -148.481,A -90.000,B 90.000,C 0.000} C_DIS
LIN {X 90.562,Y -36.017,Z -148.790,A -90.000,B 90.000,C 0.000} C_DIS
LIN {X 90.433,Y -36.011,Z -149.714,A -90.000,B 90.000,C 0.000} C_DIS
LIN {X 90.095,Y -36.006,Z -152.051,A -90.000,B 90.000,C 0.000} C_DIS
LIN {X 90.012,Y -36.005,Z -152.611,A -90.000,B 90.000,C 0.000} C_DIS
LIN {X 89.912,Y -36.000,Z -153.203,A -90.000,B 90.000,C 0.000} C_DIS
LIN {X 89.818,Y -35.997,Z -153.749,A -90.000,B 90.000,C 0.000} C_DIS
LIN {X 89.550,Y -35.995,Z -155.273,A -90.000,B 90.000,C 0.000} C_DIS
LIN {X 89.368,Y -35.991,Z -156.289,A -90.000,B 90.000,C 0.000} C_DIS
LIN {X 89.320,Y -35.986,Z -156.538,A -90.000,B 90.000,C 0.000} C_DIS
LIN {X 89.146,Y -35.982,Z -157.392,A -90.000,B 90.000,C 0.000} C_DIS
LIN {X 88.840,Y -35.981,Z -158.854,A -90.000,B 90.000,C 0.000} C_DIS
LIN {X 88.614,Y -35.977,Z -159.923,A -90.000,B 90.000,C 0.000} C_DIS
LIN {X 88.541,Y -35.971,Z -160.244,A -90.000,B 90.000,C 0.000} C_DIS
LIN {X 88.351,Y -35.969,Z -161.037,A -90.000,B 90.000,C 0.000} C_DIS
LIN {X 88.007,Y -35.969,Z -162.455,A -90.000,B 90.000,C 0.000} C_DIS
LIN {X 87.744,Y -35.967,Z -163.525,A -90.000,B 90.000,C 0.000} C_DIS
LIN {X 87.644,Y -35.962,Z -163.913,A -90.000,B 90.000,C 0.000} C_DIS
LIN {X 87.128,Y -35.961,Z -165.779,A -90.000,B 90.000,C 0.000} C_DIS
LIN {X 86.651,Y -35.963,Z -167.491,A -90.000,B 90.000,C 0.000} C_DIS
LIN {X 86.526,Y -35.959,Z -167.920,A -90.000,B 90.000,C 0.000} C_DIS
LIN {X 86.090,Y -35.961,Z -169.369,A -90.000,B 90.000,C 0.000} C_DIS
LIN {X 85.601,Y -35.964,Z -170.986,A -90.000,B 90.000,C 0.000} C_DIS
LIN {X 85.441,Y -35.963,Z -171.500,A -90.000,B 90.000,C 0.000} C_DIS
LIN {X 84.674,Y -35.966,Z -173.934,A -90.000,B 90.000,C 0.000} C_DIS
LIN {X 84.365,Y -35.966,Z -174.912,A -90.000,B 90.000,C 0.000} C_DIS
LIN {X 83.950,Y -35.963,Z -176.231,A -90.000,B 90.000,C 0.000} C_DIS
LIN {X 83.412,Y -35.963,Z -177.920,A -90.000,B 90.000,C 0.000} C_DIS
LIN {X 82.987,Y -35.962,Z -179.303,A -90.000,B 90.000,C 0.000} C_DIS
LIN {X 82.555,Y -35.951,Z -180.743,A -90.000,B 90.000,C 0.000} C_DIS
LIN {X 82.118,Y -35.948,Z -182.201,A -90.000,B 90.000,C 0.000} C_DIS
LIN {X 81.859,Y -35.937,Z -183.092,A -90.000,B 90.000,C 0.000} C_DIS
LIN {X 81.740,Y -35.931,Z -183.497,A -90.000,B 90.000,C 0.000} C_DIS
LIN {X 81.292,Y -35.927,Z -185.001,A -90.000,B 90.000,C 0.000} C_DIS
LIN {X 81.087,Y -35.916,Z -185.716,A -90.000,B 90.000,C 0.000} C_DIS
LIN {X 80.967,Y -35.908,Z -186.121,A -90.000,B 90.000,C 0.000} C_DIS
LIN {X 80.490,Y -35.902,Z -187.712,A -90.000,B 90.000,C 0.000} C_DIS
LIN {X 80.338,Y -35.895,Z -188.236,A -90.000,B 90.000,C 0.000} C_DIS
LIN {X 80.205,Y -35.885,Z -188.678,A -90.000,B 90.000,C 0.000} C_DIS
LIN {X 79.688,Y -35.880,Z -190.360,A -90.000,B 90.000,C 0.000} C_DIS
LIN {X 79.588,Y -35.875,Z -190.696,A -90.000,B 90.000,C 0.000} C_DIS
LIN {X 79.455,Y -35.866,Z -191.123,A -90.000,B 90.000,C 0.000} C_DIS
LIN {X 78.837,Y -35.861,Z -193.033,A -90.000,B 90.000,C 0.000} C_DIS
LIN {X 78.635,Y -35.852,Z -193.669,A -90.000,B 90.000,C 0.000} C_DIS
LIN {X 78.028,Y -35.848,Z -195.437,A -90.000,B 90.000,C 0.000} C_DIS
LIN {X 77.839,Y -35.847,Z -195.989,A -90.000,B 90.000,C 0.000} C_DIS
LIN {X 77.641,Y -35.842,Z -196.575,A -90.000,B 90.000,C 0.000} C_DIS
LIN {X 76.657,Y -35.839,Z -199.285,A -90.000,B 90.000,C 0.000} C_DIS
LIN {X 76.418,Y -35.836,Z -199.946,A -90.000,B 90.000,C 0.000} C_DIS
LIN {X 75.159,Y -35.834,Z -203.265,A -90.000,B 90.000,C 0.000} C_DIS
LIN {X 74.969,Y -35.833,Z -203.766,A -90.000,B 90.000,C 0.000} C_DIS
LIN {X 74.854,Y -35.831,Z -204.063,A -90.000,B 90.000,C 0.000} C_DIS
LIN {X 74.354,Y -35.832,Z -205.330,A -90.000,B 90.000,C 0.000} C_DIS
LIN {X 73.217,Y -35.830,Z -208.201,A -90.000,B 90.000,C 0.000} C_DIS
LIN {X 73.096,Y -35.829,Z -208.502,A -90.000,B 90.000,C 0.000} C_DIS
LIN {X 72.490,Y -35.831,Z -209.978,A -90.000,B 90.000,C 0.000} C_DIS
LIN {X 71.217,Y -35.830,Z -213.065,A -90.000,B 90.000,C 0.000} C_DIS
LIN {X 71.104,Y -35.829,Z -213.333,A -90.000,B 90.000,C 0.000} C_DIS
LIN {X 70.407,Y -35.832,Z -214.965,A -90.000,B 90.000,C 0.000} C_DIS
LIN {X 69.043,Y -35.831,Z -218.136,A -90.000,B 90.000,C 0.000} C_DIS
LIN {X 68.927,Y -35.829,Z -218.398,A -90.000,B 90.000,C 0.000} C_DIS
LIN {X 67.700,Y -35.828,Z -221.125,A -90.000,B 90.000,C 0.000} C_DIS
LIN {X 66.725,Y -35.833,Z -223.307,A -90.000,B 90.000,C 0.000} C_DIS
LIN {X 66.542,Y -35.830,Z -223.702,A -90.000,B 90.000,C 0.000} C_DIS
LIN {X 66.004,Y -35.832,Z -224.840,A -90.000,B 90.000,C 0.000} C_DIS
LIN {X 65.315,Y -35.831,Z -226.303,A -90.000,B 90.000,C 0.000} C_DIS
LIN {X 64.167,Y -35.841,Z -228.768,A -90.000,B 90.000,C 0.000} C_DIS
LIN {X 64.030,Y -35.840,Z -229.058,A -90.000,B 90.000,C 0.000} C_DIS
LIN {X 63.898,Y -35.839,Z -229.328,A -90.000,B 90.000,C 0.000} C_DIS
LIN {X 63.640,Y -35.842,Z -229.842,A -90.000,B 90.000,C 0.000} C_DIS
LIN {X 62.662,Y -35.842,Z -231.826,A -90.000,B 90.000,C 0.000} C_DIS
LIN {X 61.439,Y -35.862,Z -234.357,A -90.000,B 90.000,C 0.000} C_DIS
LIN {X 61.367,Y -35.861,Z -234.499,A -90.000,B 90.000,C 0.000} C_DIS
LIN {X 61.202,Y -35.864,Z -234.810,A -90.000,B 90.000,C 0.000} C_DIS
LIN {X 60.382,Y -35.863,Z -236.397,A -90.000,B 90.000,C 0.000} C_DIS
LIN {X 58.773,Y -35.909,Z -239.611,A -90.000,B 90.000,C 0.000} C_DIS
LIN {X 58.591,Y -35.913,Z -239.972,A -90.000,B 90.000,C 0.000} C_DIS
LIN {X 56.946,Y -35.985,Z -243.139,A -90.000,B 90.000,C 0.000} C_DIS
LIN {X 56.717,Y -35.985,Z -243.561,A -90.000,B 90.000,C 0.000} C_DIS
LIN {X 56.717,Y -60.000,Z -243.561,A -90.000,B 90.000,C 0.000} C_DIS
LIN {X -90.766,Y -60.000,Z -243.561,A -90.000,B 90.000,C 0.000} C_DIS
LIN {X -90.766,Y -36.495,Z -243.561,A -90.000,B 90.000,C 0.000} C_DIS
LIN {X -90.622,Y -36.299,Z -243.178,A -90.000,B 90.000,C 0.000} C_DIS
LIN {X -90.285,Y -36.118,Z -242.684,A -90.000,B 90.000,C 0.000} C_DIS
LIN {X -89.911,Y -36.058,Z -242.340,A -90.000,B 90.000,C 0.000} C_DIS
LIN {X -89.817,Y -36.056,Z -242.273,A -90.000,B 90.000,C 0.000} C_DIS
LIN {X -88.839,Y -36.058,Z -241.605,A -90.000,B 90.000,C 0.000} C_DIS
LIN {X -86.768,Y -36.081,Z -240.217,A -90.000,B 90.000,C 0.000} C_DIS
LIN {X -86.581,Y -36.081,Z -240.094,A -90.000,B 90.000,C 0.000} C_DIS
LIN {X -85.936,Y -36.077,Z -239.672,A -90.000,B 90.000,C 0.000} C_DIS
LIN {X -85.368,Y -36.080,Z -239.313,A -90.000,B 90.000,C 0.000} C_DIS
LIN {X -82.414,Y -36.091,Z -237.453,A -90.000,B 90.000,C 0.000} C_DIS
LIN {X -79.383,Y -36.126,Z -235.578,A -90.000,B 90.000,C 0.000} C_DIS
LIN {X -78.773,Y -36.131,Z -235.203,A -90.000,B 90.000,C 0.000} C_DIS
LIN {X -78.595,Y -36.131,Z -235.095,A -90.000,B 90.000,C 0.000} C_DIS
LIN {X -77.715,Y -36.119,Z -234.571,A -90.000,B 90.000,C 0.000} C_DIS
LIN {X -76.071,Y -36.119,Z -233.628,A -90.000,B 90.000,C 0.000} C_DIS
LIN {X -72.326,Y -36.134,Z -231.503,A -90.000,B 90.000,C 0.000} C_DIS
LIN {X -71.657,Y -36.134,Z -231.126,A -90.000,B 90.000,C 0.000} C_DIS
LIN {X -70.067,Y -36.139,Z -230.236,A -90.000,B 90.000,C 0.000} C_DIS
LIN {X -69.362,Y -36.131,Z -229.854,A -90.000,B 90.000,C 0.000} C_DIS
LIN {X -69.158,Y -36.130,Z -229.746,A -90.000,B 90.000,C 0.000} C_DIS
LIN {X -61.370,Y -36.161,Z -225.710,A -90.000,B 90.000,C 0.000} C_DIS
LIN {X -60.445,Y -36.157,Z -225.237,A -90.000,B 90.000,C 0.000} C_DIS
LIN {X -55.947,Y -36.162,Z -222.991,A -90.000,B 90.000,C 0.000} C_DIS
LIN {X -53.530,Y -36.158,Z -221.791,A -90.000,B 90.000,C 0.000} C_DIS
LIN {X -50.848,Y -36.157,Z -220.466,A -90.000,B 90.000,C 0.000} C_DIS
LIN {X -50.068,Y -36.156,Z -220.082,A -90.000,B 90.000,C 0.000} C_DIS
LIN {X -44.738,Y -36.150,Z -217.477,A -90.000,B 90.000,C 0.000} C_DIS
LIN {X -44.201,Y -36.153,Z -217.212,A -90.000,B 90.000,C 0.000} C_DIS
LIN {X -43.412,Y -36.153,Z -216.815,A -90.000,B 90.000,C 0.000} C_DIS
LIN {X -41.231,Y -36.155,Z -215.722,A -90.000,B 90.000,C 0.000} C_DIS
LIN {X -38.779,Y -36.161,Z -214.498,A -90.000,B 90.000,C 0.000} C_DIS
LIN {X -37.895,Y -36.160,Z -214.059,A -90.000,B 90.000,C 0.000} C_DIS
LIN {X -37.094,Y -36.172,Z -213.652,A -90.000,B 90.000,C 0.000} C_DIS
LIN {X -36.899,Y -36.174,Z -213.550,A -90.000,B 90.000,C 0.000} C_DIS
LIN {X -36.052,Y -36.174,Z -213.111,A -90.000,B 90.000,C 0.000} C_DIS
LIN {X -33.399,Y -36.162,Z -211.716,A -90.000,B 90.000,C 0.000} C_DIS
LIN {X -32.325,Y -36.162,Z -211.148,A -90.000,B 90.000,C 0.000} C_DIS
LIN {X -31.628,Y -36.170,Z -210.776,A -90.000,B 90.000,C 0.000} C_DIS
LIN {X -29.733,Y -36.167,Z -209.723,A -90.000,B 90.000,C 0.000} C_DIS
LIN {X -27.395,Y -36.182,Z -208.432,A -90.000,B 90.000,C 0.000} C_DIS
LIN {X -26.875,Y -36.190,Z -208.135,A -90.000,B 90.000,C 0.000} C_DIS
LIN {X -25.918,Y -36.193,Z -207.566,A -90.000,B 90.000,C 0.000} C_DIS
LIN {X -24.097,Y -36.205,Z -206.475,A -90.000,B 90.000,C 0.000} C_DIS
LIN {X -23.117,Y -36.206,Z -205.878,A -90.000,B 90.000,C 0.000} C_DIS
LIN {X -22.605,Y -36.215,Z -205.559,A -90.000,B 90.000,C 0.000} C_DIS
LIN {X -20.846,Y -36.226,Z -204.403,A -90.000,B 90.000,C 0.000} C_DIS
LIN {X -19.452,Y -36.225,Z -203.474,A -90.000,B 90.000,C 0.000} C_DIS
LIN {X -18.719,Y -36.241,Z -202.973,A -90.000,B 90.000,C 0.000} C_DIS
LIN {X -16.073,Y -36.242,Z -201.057,A -90.000,B 90.000,C 0.000} C_DIS
LIN {X -15.284,Y -36.258,Z -200.477,A -90.000,B 90.000,C 0.000} C_DIS
LIN {X -12.575,Y -36.255,Z -198.375,A -90.000,B 90.000,C 0.000} C_DIS
LIN {X -11.801,Y -36.266,Z -197.766,A -90.000,B 90.000,C 0.000} C_DIS
LIN {X -10.110,Y -36.263,Z -196.379,A -90.000,B 90.000,C 0.000} C_DIS
LIN {X -9.038,Y -36.264,Z -195.505,A -90.000,B 90.000,C 0.000} C_DIS
LIN {X -8.262,Y -36.274,Z -194.866,A -90.000,B 90.000,C 0.000} C_DIS
LIN {X -5.423,Y -36.269,Z -192.464,A -90.000,B 90.000,C 0.000} C_DIS
LIN {X -4.648,Y -36.271,Z -191.806,A -90.000,B 90.000,C 0.000} C_DIS
LIN {X -2.857,Y -36.263,Z -190.264,A -90.000,B 90.000,C 0.000} C_DIS
LIN {X -1.777,Y -36.267,Z -189.327,A -90.000,B 90.000,C 0.000} C_DIS
LIN {X -0.911,Y -36.257,Z -188.551,A -90.000,B 90.000,C 0.000} C_DIS
LIN {X 0.550,Y -36.248,Z -187.266,A -90.000,B 90.000,C 0.000} C_DIS
LIN {X 1.573,Y -36.252,Z -186.358,A -90.000,B 90.000,C 0.000} C_DIS
LIN {X 2.791,Y -36.235,Z -185.235,A -90.000,B 90.000,C 0.000} C_DIS
LIN {X 3.841,Y -36.229,Z -184.289,A -90.000,B 90.000,C 0.000} C_DIS
LIN {X 4.853,Y -36.232,Z -183.371,A -90.000,B 90.000,C 0.000} C_DIS
LIN {X 6.300,Y -36.215,Z -182.010,A -90.000,B 90.000,C 0.000} C_DIS
LIN {X 7.074,Y -36.214,Z -181.295,A -90.000,B 90.000,C 0.000} C_DIS
LIN {X 7.968,Y -36.215,Z -180.465,A -90.000,B 90.000,C 0.000} C_DIS
LIN {X 8.839,Y -36.207,Z -179.640,A -90.000,B 90.000,C 0.000} C_DIS
LIN {X 9.483,Y -36.206,Z -179.026,A -90.000,B 90.000,C 0.000} C_DIS
LIN {X 10.422,Y -36.207,Z -178.140,A -90.000,B 90.000,C 0.000} C_DIS
LIN {X 11.482,Y -36.215,Z -177.129,A -90.000,B 90.000,C 0.000} C_DIS
LIN {X 12.220,Y -36.226,Z -176.422,A -90.000,B 90.000,C 0.000} C_DIS
LIN {X 12.732,Y -36.231,Z -175.928,A -90.000,B 90.000,C 0.000} C_DIS
LIN {X 13.320,Y -36.249,Z -175.353,A -90.000,B 90.000,C 0.000} C_DIS
LIN {X 13.706,Y -36.255,Z -174.964,A -90.000,B 90.000,C 0.000} C_DIS
LIN {X 14.878,Y -36.281,Z -173.781,A -90.000,B 90.000,C 0.000} C_DIS
LIN {X 15.200,Y -36.297,Z -173.448,A -90.000,B 90.000,C 0.000} C_DIS
LIN {X 16.300,Y -36.331,Z -172.246,A -90.000,B 90.000,C 0.000} C_DIS
LIN {X 16.848,Y -36.370,Z -171.626,A -90.000,B 90.000,C 0.000} C_DIS
LIN {X 17.618,Y -36.403,Z -170.681,A -90.000,B 90.000,C 0.000} C_DIS
LIN {X 17.838,Y -36.422,Z -170.400,A -90.000,B 90.000,C 0.000} C_DIS
LIN {X 18.718,Y -36.475,Z -169.147,A -90.000,B 90.000,C 0.000} C_DIS
LIN {X 19.048,Y -36.535,Z -168.648,A -90.000,B 90.000,C 0.000} C_DIS
LIN {X 19.293,Y -36.573,Z -168.240,A -90.000,B 90.000,C 0.000} C_DIS
LIN {X 19.812,Y -36.627,Z -167.397,A -90.000,B 90.000,C 0.000} C_DIS
LIN {X 20.031,Y -36.636,Z -166.928,A -90.000,B 90.000,C 0.000} C_DIS
LIN {X 20.097,Y -36.649,Z -166.794,A -90.000,B 90.000,C 0.000} C_DIS
LIN {X 20.218,Y -36.673,Z -166.565,A -90.000,B 90.000,C 0.000} C_DIS
LIN {X 20.467,Y -36.746,Z -166.083,A -90.000,B 90.000,C 0.000} C_DIS
LIN {X 20.619,Y -36.796,Z -165.637,A -90.000,B 90.000,C 0.000} C_DIS
LIN {X 20.709,Y -36.833,Z -165.188,A -90.000,B 90.000,C 0.000} C_DIS
LIN {X 20.718,Y -36.842,Z -165.006,A -90.000,B 90.000,C 0.000} C_DIS
LIN {X 20.641,Y -36.830,Z -164.853,A -90.000,B 90.000,C 0.000} C_DIS
LIN {X 20.597,Y -36.822,Z -164.746,A -90.000,B 90.000,C 0.000} C_DIS
LIN {X 20.508,Y -36.802,Z -164.481,A -90.000,B 90.000,C 0.000} C_DIS
LIN {X 20.450,Y -36.806,Z -164.303,A -90.000,B 90.000,C 0.000} C_DIS
LIN {X 20.415,Y -36.801,Z -164.266,A -90.000,B 90.000,C 0.000} C_DIS
LIN {X 20.211,Y -36.773,Z -164.042,A -90.000,B 90.000,C 0.000} C_DIS
LIN {X 20.106,Y -36.760,Z -163.916,A -90.000,B 90.000,C 0.000} C_DIS
LIN {X 19.990,Y -36.749,Z -163.748,A -90.000,B 90.000,C 0.000} C_DIS
LIN {X 19.882,Y -36.741,Z -163.567,A -90.000,B 90.000,C 0.000} C_DIS
LIN {X 19.808,Y -36.744,Z -163.446,A -90.000,B 90.000,C 0.000} C_DIS
LIN {X 19.739,Y -36.750,Z -163.313,A -90.000,B 90.000,C 0.000} C_DIS
LIN {X 19.684,Y -36.755,Z -163.199,A -90.000,B 90.000,C 0.000} C_DIS
LIN {X 19.551,Y -36.742,Z -163.034,A -90.000,B 90.000,C 0.000} C_DIS
LIN {X 19.205,Y -36.700,Z -162.598,A -90.000,B 90.000,C 0.000} C_DIS
LIN {X 19.148,Y -36.693,Z -162.523,A -90.000,B 90.000,C 0.000} C_DIS
LIN {X 18.824,Y -36.664,Z -162.043,A -90.000,B 90.000,C 0.000} C_DIS
LIN {X 18.745,Y -36.653,Z -161.902,A -90.000,B 90.000,C 0.000} C_DIS
LIN {X 18.625,Y -36.640,Z -161.668,A -90.000,B 90.000,C 0.000} C_DIS
LIN {X 18.583,Y -36.635,Z -161.583,A -90.000,B 90.000,C 0.000} C_DIS
LIN {X 18.503,Y -36.628,Z -161.408,A -90.000,B 90.000,C 0.000} C_DIS
LIN {X 18.341,Y -36.610,Z -161.094,A -90.000,B 90.000,C 0.000} C_DIS
LIN {X 18.296,Y -36.610,Z -161.010,A -90.000,B 90.000,C 0.000} C_DIS
LIN {X 18.079,Y -36.618,Z -160.565,A -90.000,B 90.000,C 0.000} C_DIS
LIN {X 17.882,Y -36.597,Z -160.135,A -90.000,B 90.000,C 0.000} C_DIS
LIN {X 17.828,Y -36.592,Z -160.007,A -90.000,B 90.000,C 0.000} C_DIS
LIN {X 17.745,Y -36.589,Z -159.777,A -90.000,B 90.000,C 0.000} C_DIS
LIN {X 17.670,Y -36.594,Z -159.550,A -90.000,B 90.000,C 0.000} C_DIS
LIN {X 17.629,Y -36.598,Z -159.423,A -90.000,B 90.000,C 0.000} C_DIS
LIN {X 17.470,Y -36.619,Z -158.884,A -90.000,B 90.000,C 0.000} C_DIS
LIN {X 17.288,Y -36.633,Z -158.254,A -90.000,B 90.000,C 0.000} C_DIS
LIN {X 17.127,Y -36.632,Z -157.743,A -90.000,B 90.000,C 0.000} C_DIS
LIN {X 17.082,Y -36.636,Z -157.565,A -90.000,B 90.000,C 0.000} C_DIS
LIN {X 17.002,Y -36.651,Z -157.172,A -90.000,B 90.000,C 0.000} C_DIS
LIN {X 16.904,Y -36.673,Z -156.696,A -90.000,B 90.000,C 0.000} C_DIS
LIN {X 16.891,Y -36.674,Z -156.629,A -90.000,B 90.000,C 0.000} C_DIS
LIN {X 16.864,Y -36.677,Z -156.461,A -90.000,B 90.000,C 0.000} C_DIS
LIN {X 16.835,Y -36.677,Z -156.254,A -90.000,B 90.000,C 0.000} C_DIS
LIN {X 16.726,Y -36.681,Z -155.309,A -90.000,B 90.000,C 0.000} C_DIS
LIN {X 16.681,Y -36.681,Z -154.936,A -90.000,B 90.000,C 0.000} C_DIS
LIN {X 16.663,Y -36.672,Z -154.761,A -90.000,B 90.000,C 0.000} C_DIS
LIN {X 16.658,Y -36.670,Z -154.681,A -90.000,B 90.000,C 0.000} C_DIS
LIN {X 16.657,Y -36.667,Z -154.577,A -90.000,B 90.000,C 0.000} C_DIS
LIN {X 16.673,Y -36.662,Z -154.207,A -90.000,B 90.000,C 0.000} C_DIS
LIN {X 16.764,Y -36.632,Z -153.173,A -90.000,B 90.000,C 0.000} C_DIS
LIN {X 16.787,Y -36.636,Z -153.014,A -90.000,B 90.000,C 0.000} C_DIS
LIN {X 16.858,Y -36.648,Z -152.591,A -90.000,B 90.000,C 0.000} C_DIS
LIN {X 16.909,Y -36.655,Z -152.335,A -90.000,B 90.000,C 0.000} C_DIS
LIN {X 16.939,Y -36.657,Z -152.194,A -90.000,B 90.000,C 0.000} C_DIS
LIN {X 16.983,Y -36.660,Z -152.027,A -90.000,B 90.000,C 0.000} C_DIS
LIN {X 17.043,Y -36.667,Z -151.853,A -90.000,B 90.000,C 0.000} C_DIS
LIN {X 16.717,Y -36.573,Z -151.924,A -90.000,B 90.000,C 0.000} C_DIS
LIN {X 16.340,Y -36.463,Z -151.998,A -90.000,B 90.000,C 0.000} C_DIS
LIN {X 15.970,Y -36.354,Z -152.062,A -90.000,B 90.000,C 0.000} C_DIS
LIN {X 15.852,Y -36.319,Z -152.079,A -90.000,B 90.000,C 0.000} C_DIS
LIN {X 15.305,Y -36.209,Z -152.181,A -90.000,B 90.000,C 0.000} C_DIS
LIN {X 14.840,Y -36.116,Z -152.260,A -90.000,B 90.000,C 0.000} C_DIS
LIN {X 14.467,Y -36.041,Z -152.305,A -90.000,B 90.000,C 0.000} C_DIS
LIN {X 14.226,Y -36.011,Z -152.346,A -90.000,B 90.000,C 0.000} C_DIS
LIN {X 13.935,Y -35.964,Z -152.385,A -90.000,B 90.000,C 0.000} C_DIS
LIN {X 13.603,Y -35.911,Z -152.422,A -90.000,B 90.000,C 0.000} C_DIS
LIN {X 13.167,Y -35.843,Z -152.464,A -90.000,B 90.000,C 0.000} C_DIS
LIN {X 12.524,Y -35.743,Z -152.504,A -90.000,B 90.000,C 0.000} C_DIS
LIN {X 11.580,Y -35.667,Z -152.631,A -90.000,B 90.000,C 0.000} C_DIS
LIN {X 11.050,Y -35.662,Z -152.751,A -90.000,B 90.000,C 0.000} C_DIS
LIN {X 10.392,Y -35.660,Z -152.896,A -90.000,B 90.000,C 0.000} C_DIS
LIN {X 10.307,Y -35.661,Z -152.914,A -90.000,B 90.000,C 0.000} C_DIS
LIN {X 9.823,Y -35.669,Z -153.000,A -90.000,B 90.000,C 0.000} C_DIS
LIN {X 9.289,Y -35.660,Z -153.071,A -90.000,B 90.000,C 0.000} C_DIS
LIN {X 7.618,Y -35.648,Z -153.316,A -90.000,B 90.000,C 0.000} C_DIS
LIN {X 7.191,Y -35.657,Z -153.375,A -90.000,B 90.000,C 0.000} C_DIS
LIN {X 6.770,Y -35.667,Z -153.413,A -90.000,B 90.000,C 0.000} C_DIS
LIN {X 6.237,Y -35.664,Z -153.435,A -90.000,B 90.000,C 0.000} C_DIS
LIN {X 4.472,Y -35.642,Z -153.512,A -90.000,B 90.000,C 0.000} C_DIS
LIN {X 4.175,Y -35.640,Z -153.527,A -90.000,B 90.000,C 0.000} C_DIS
LIN {X 3.902,Y -35.646,Z -153.537,A -90.000,B 90.000,C 0.000} C_DIS
LIN {X 3.819,Y -35.646,Z -153.536,A -90.000,B 90.000,C 0.000} C_DIS
LIN {X 3.658,Y -35.646,Z -153.535,A -90.000,B 90.000,C 0.000} C_DIS
LIN {X 3.461,Y -35.650,Z -153.531,A -90.000,B 90.000,C 0.000} C_DIS
LIN {X 2.151,Y -35.638,Z -153.434,A -90.000,B 90.000,C 0.000} C_DIS
LIN {X 1.027,Y -35.621,Z -153.355,A -90.000,B 90.000,C 0.000} C_DIS
LIN {X 0.443,Y -35.616,Z -153.321,A -90.000,B 90.000,C 0.000} C_DIS
LIN {X 0.238,Y -35.620,Z -153.305,A -90.000,B 90.000,C 0.000} C_DIS
LIN {X -0.044,Y -35.615,Z -153.264,A -90.000,B 90.000,C 0.000} C_DIS
LIN {X -0.216,Y -35.616,Z -153.237,A -90.000,B 90.000,C 0.000} C_DIS
LIN {X -2.413,Y -35.600,Z -152.817,A -90.000,B 90.000,C 0.000} C_DIS
LIN {X -3.523,Y -35.595,Z -152.617,A -90.000,B 90.000,C 0.000} C_DIS
LIN {X -3.660,Y -35.591,Z -152.582,A -90.000,B 90.000,C 0.000} C_DIS
LIN {X -3.968,Y -35.588,Z -152.499,A -90.000,B 90.000,C 0.000} C_DIS
LIN {X -6.782,Y -35.576,Z -151.654,A -90.000,B 90.000,C 0.000} C_DIS
LIN {X -7.459,Y -35.575,Z -151.455,A -90.000,B 90.000,C 0.000} C_DIS
LIN {X -7.682,Y -35.565,Z -151.372,A -90.000,B 90.000,C 0.000} C_DIS
LIN {X -7.767,Y -35.564,Z -151.340,A -90.000,B 90.000,C 0.000} C_DIS
LIN {X -8.199,Y -35.562,Z -151.166,A -90.000,B 90.000,C 0.000} C_DIS
LIN {X -11.468,Y -35.563,Z -149.832,A -90.000,B 90.000,C 0.000} C_DIS
LIN {X -11.787,Y -35.549,Z -149.675,A -90.000,B 90.000,C 0.000} C_DIS
LIN {X -11.870,Y -35.547,Z -149.632,A -90.000,B 90.000,C 0.000} C_DIS
LIN {X -12.905,Y -35.549,Z -149.089,A -90.000,B 90.000,C 0.000} C_DIS
LIN {X -14.957,Y -35.556,Z -148.016,A -90.000,B 90.000,C 0.000} C_DIS
LIN {X -15.597,Y -35.557,Z -147.679,A -90.000,B 90.000,C 0.000} C_DIS
LIN {X -15.843,Y -35.546,Z -147.525,A -90.000,B 90.000,C 0.000} C_DIS
LIN {X -16.018,Y -35.544,Z -147.411,A -90.000,B 90.000,C 0.000} C_DIS
LIN {X -17.210,Y -35.555,Z -146.637,A -90.000,B 90.000,C 0.000} C_DIS
LIN {X -19.163,Y -35.568,Z -145.356,A -90.000,B 90.000,C 0.000} C_DIS
LIN {X -19.544,Y -35.566,Z -145.099,A -90.000,B 90.000,C 0.000} C_DIS
LIN {X -19.712,Y -35.559,Z -144.972,A -90.000,B 90.000,C 0.000} C_DIS
LIN {X -20.006,Y -35.549,Z -144.747,A -90.000,B 90.000,C 0.000} C_DIS
LIN {X -20.476,Y -35.552,Z -144.375,A -90.000,B 90.000,C 0.000} C_DIS
LIN {X -21.691,Y -35.553,Z -143.414,A -90.000,B 90.000,C 0.000} C_DIS
LIN {X -23.073,Y -35.566,Z -142.334,A -90.000,B 90.000,C 0.000} C_DIS
LIN {X -23.406,Y -35.563,Z -142.056,A -90.000,B 90.000,C 0.000} C_DIS
LIN {X -23.642,Y -35.557,Z -141.845,A -90.000,B 90.000,C 0.000} C_DIS
LIN {X -24.268,Y -35.564,Z -141.262,A -90.000,B 90.000,C 0.000} C_DIS
LIN {X -25.519,Y -35.595,Z -140.083,A -90.000,B 90.000,C 0.000} C_DIS
LIN {X -26.095,Y -35.607,Z -139.531,A -90.000,B 90.000,C 0.000} C_DIS
LIN {X -26.510,Y -35.617,Z -139.136,A -90.000,B 90.000,C 0.000} C_DIS
LIN {X -26.823,Y -35.612,Z -138.806,A -90.000,B 90.000,C 0.000} C_DIS
LIN {X -27.014,Y -35.608,Z -138.597,A -90.000,B 90.000,C 0.000} C_DIS
LIN {X -28.073,Y -35.637,Z -137.389,A -90.000,B 90.000,C 0.000} C_DIS
LIN {X -28.900,Y -35.661,Z -136.449,A -90.000,B 90.000,C 0.000} C_DIS
LIN {X -29.505,Y -35.681,Z -135.760,A -90.000,B 90.000,C 0.000} C_DIS
LIN {X -29.593,Y -35.678,Z -135.646,A -90.000,B 90.000,C 0.000} C_DIS
LIN {X -29.756,Y -35.676,Z -135.430,A -90.000,B 90.000,C 0.000} C_DIS
LIN {X -29.862,Y -35.676,Z -135.288,A -90.000,B 90.000,C 0.000} C_DIS
LIN {X -30.111,Y -35.685,Z -134.937,A -90.000,B 90.000,C 0.000} C_DIS
LIN {X -30.775,Y -35.699,Z -133.975,A -90.000,B 90.000,C 0.000} C_DIS
LIN {X -31.210,Y -35.711,Z -133.342,A -90.000,B 90.000,C 0.000} C_DIS
LIN {X -31.547,Y -35.725,Z -132.845,A -90.000,B 90.000,C 0.000} C_DIS
LIN {X -31.837,Y -35.733,Z -132.407,A -90.000,B 90.000,C 0.000} C_DIS
LIN {X -31.968,Y -35.730,Z -132.193,A -90.000,B 90.000,C 0.000} C_DIS
LIN {X -32.061,Y -35.732,Z -132.037,A -90.000,B 90.000,C 0.000} C_DIS
LIN {X -32.161,Y -35.732,Z -131.857,A -90.000,B 90.000,C 0.000} C_DIS
LIN {X -32.752,Y -35.748,Z -130.767,A -90.000,B 90.000,C 0.000} C_DIS
LIN {X -33.698,Y -35.781,Z -129.006,A -90.000,B 90.000,C 0.000} C_DIS
LIN {X -33.790,Y -35.778,Z -128.812,A -90.000,B 90.000,C 0.000} C_DIS
LIN {X -34.184,Y -35.782,Z -127.937,A -90.000,B 90.000,C 0.000} C_DIS
LIN {X -35.000,Y -35.800,Z -126.097,A -90.000,B 90.000,C 0.000} C_DIS
LIN {X -35.159,Y -35.806,Z -125.734,A -90.000,B 90.000,C 0.000} C_DIS
LIN {X -35.167,Y -35.805,Z -125.712,A -90.000,B 90.000,C 0.000} C_DIS
LIN {X -35.607,Y -35.802,Z -124.494,A -90.000,B 90.000,C 0.000} C_DIS
LIN {X -36.086,Y -35.803,Z -123.170,A -90.000,B 90.000,C 0.000} C_DIS
LIN {X -36.146,Y -35.808,Z -122.994,A -90.000,B 90.000,C 0.000} C_DIS
LIN {X -36.276,Y -35.817,Z -122.576,A -90.000,B 90.000,C 0.000} C_DIS
LIN {X -36.352,Y -35.816,Z -122.309,A -90.000,B 90.000,C 0.000} C_DIS
LIN {X -36.607,Y -35.801,Z -121.444,A -90.000,B 90.000,C 0.000} C_DIS
LIN {X -36.872,Y -35.793,Z -120.581,A -90.000,B 90.000,C 0.000} C_DIS
LIN {X -37.007,Y -35.798,Z -120.119,A -90.000,B 90.000,C 0.000} C_DIS
LIN {X -37.061,Y -35.806,Z -119.917,A -90.000,B 90.000,C 0.000} C_DIS
LIN {X -37.130,Y -35.809,Z -119.678,A -90.000,B 90.000,C 0.000} C_DIS
LIN {X -37.228,Y -35.800,Z -119.282,A -90.000,B 90.000,C 0.000} C_DIS
LIN {X -37.590,Y -35.797,Z -117.692,A -90.000,B 90.000,C 0.000} C_DIS
LIN {X -37.653,Y -35.794,Z -117.396,A -90.000,B 90.000,C 0.000} C_DIS
LIN {X -37.734,Y -35.808,Z -116.945,A -90.000,B 90.000,C 0.000} C_DIS
LIN {X -37.824,Y -35.825,Z -116.451,A -90.000,B 90.000,C 0.000} C_DIS
LIN {X -37.882,Y -35.820,Z -116.003,A -90.000,B 90.000,C 0.000} C_DIS
LIN {X -38.049,Y -35.778,Z -114.884,A -90.000,B 90.000,C 0.000} C_DIS
LIN {X -38.141,Y -35.765,Z -114.317,A -90.000,B 90.000,C 0.000} C_DIS
LIN {X -38.210,Y -35.763,Z -113.852,A -90.000,B 90.000,C 0.000} C_DIS
LIN {X -38.245,Y -35.767,Z -113.592,A -90.000,B 90.000,C 0.000} C_DIS
LIN {X -38.272,Y -35.775,Z -113.364,A -90.000,B 90.000,C 0.000} C_DIS
LIN {X -38.323,Y -35.781,Z -112.787,A -90.000,B 90.000,C 0.000} C_DIS
LIN {X -38.377,Y -35.772,Z -111.909,A -90.000,B 90.000,C 0.000} C_DIS
LIN {X -38.391,Y -35.766,Z -111.412,A -90.000,B 90.000,C 0.000} C_DIS
LIN {X -38.405,Y -35.755,Z -111.025,A -90.000,B 90.000,C 0.000} C_DIS
LIN {X -38.409,Y -35.758,Z -110.721,A -90.000,B 90.000,C 0.000} C_DIS
LIN {X -38.416,Y -35.770,Z -110.296,A -90.000,B 90.000,C 0.000} C_DIS
LIN {X -38.418,Y -35.789,Z -109.908,A -90.000,B 90.000,C 0.000} C_DIS
LIN {X -38.409,Y -35.794,Z -109.652,A -90.000,B 90.000,C 0.000} C_DIS
LIN {X -38.403,Y -35.796,Z -109.473,A -90.000,B 90.000,C 0.000} C_DIS
LIN {X -38.345,Y -35.769,Z -108.351,A -90.000,B 90.000,C 0.000} C_DIS
LIN {X -38.315,Y -35.760,Z -107.813,A -90.000,B 90.000,C 0.000} C_DIS
LIN {X -38.300,Y -35.757,Z -107.558,A -90.000,B 90.000,C 0.000} C_DIS
LIN {X -38.280,Y -35.761,Z -107.311,A -90.000,B 90.000,C 0.000} C_DIS
LIN {X -38.261,Y -35.768,Z -107.112,A -90.000,B 90.000,C 0.000} C_DIS
LIN {X -38.226,Y -35.783,Z -106.777,A -90.000,B 90.000,C 0.000} C_DIS
LIN {X -38.160,Y -35.790,Z -106.320,A -90.000,B 90.000,C 0.000} C_DIS
LIN {X -38.126,Y -35.787,Z -106.130,A -90.000,B 90.000,C 0.000} C_DIS
LIN {X -37.877,Y -35.777,Z -104.756,A -90.000,B 90.000,C 0.000} C_DIS
LIN {X -37.860,Y -35.778,Z -104.670,A -90.000,B 90.000,C 0.000} C_DIS
LIN {X -37.705,Y -35.799,Z -103.932,A -90.000,B 90.000,C 0.000} C_DIS
LIN {X -37.653,Y -35.803,Z -103.700,A -90.000,B 90.000,C 0.000} C_DIS
LIN {X -37.210,Y -35.800,Z -101.906,A -90.000,B 90.000,C 0.000} C_DIS
LIN {X -37.000,Y -35.819,Z -101.132,A -90.000,B 90.000,C 0.000} C_DIS
LIN {X -36.979,Y -35.869,Z -100.871,A -90.000,B 90.000,C 0.000} C_DIS
LIN {X -36.969,Y -35.911,Z -100.693,A -90.000,B 90.000,C 0.000} C_DIS
LIN {X -36.932,Y -36.024,Z -100.225,A -90.000,B 90.000,C 0.000} C_DIS
LIN {X -36.896,Y -36.109,Z -99.877,A -90.000,B 90.000,C 0.000} C_DIS
LIN {X -36.863,Y -36.179,Z -99.599,A -90.000,B 90.000,C 0.000} C_DIS
LIN {X -36.830,Y -36.241,Z -99.353,A -90.000,B 90.000,C 0.000} C_DIS
LIN {X -36.771,Y -36.346,Z -98.949,A -90.000,B 90.000,C 0.000} C_DIS
LIN {X -36.726,Y -36.431,Z -98.627,A -90.000,B 90.000,C 0.000} C_DIS
LIN {X -36.653,Y -36.561,Z -98.147,A -90.000,B 90.000,C 0.000} C_DIS
LIN {X -36.626,Y -36.605,Z -97.984,A -90.000,B 90.000,C 0.000} C_DIS
LIN {X -36.614,Y -36.627,Z -97.904,A -90.000,B 90.000,C 0.000} C_DIS
LIN {X -36.846,Y -36.626,Z -97.603,A -90.000,B 90.000,C 0.000} C_DIS
LIN {X -37.352,Y -36.633,Z -96.923,A -90.000,B 90.000,C 0.000} C_DIS
LIN {X -37.796,Y -36.633,Z -96.349,A -90.000,B 90.000,C 0.000} C_DIS
LIN {X -38.453,Y -36.611,Z -95.483,A -90.000,B 90.000,C 0.000} C_DIS
LIN {X -38.558,Y -36.609,Z -95.337,A -90.000,B 90.000,C 0.000} C_DIS
LIN {X -38.788,Y -36.609,Z -94.987,A -90.000,B 90.000,C 0.000} C_DIS
LIN {X -38.839,Y -36.610,Z -94.906,A -90.000,B 90.000,C 0.000} C_DIS
LIN {X -39.141,Y -36.620,Z -94.397,A -90.000,B 90.000,C 0.000} C_DIS
LIN {X -39.889,Y -36.614,Z -93.118,A -90.000,B 90.000,C 0.000} C_DIS
LIN {X -40.058,Y -36.617,Z -92.806,A -90.000,B 90.000,C 0.000} C_DIS
LIN {X -40.507,Y -36.635,Z -91.917,A -90.000,B 90.000,C 0.000} C_DIS
LIN {X -40.670,Y -36.640,Z -91.587,A -90.000,B 90.000,C 0.000} C_DIS
LIN {X -40.832,Y -36.641,Z -91.252,A -90.000,B 90.000,C 0.000} C_DIS
LIN {X -40.985,Y -36.634,Z -90.932,A -90.000,B 90.000,C 0.000} C_DIS
LIN {X -41.066,Y -36.634,Z -90.741,A -90.000,B 90.000,C 0.000} C_DIS
LIN {X -41.347,Y -36.648,Z -89.966,A -90.000,B 90.000,C 0.000} C_DIS
LIN {X -41.558,Y -36.663,Z -89.326,A -90.000,B 90.000,C 0.000} C_DIS
LIN {X -41.582,Y -36.666,Z -89.247,A -90.000,B 90.000,C 0.000} C_DIS
LIN {X -41.835,Y -36.699,Z -88.358,A -90.000,B 90.000,C 0.000} C_DIS
LIN {X -41.906,Y -36.704,Z -88.095,A -90.000,B 90.000,C 0.000} C_DIS
LIN {X -41.978,Y -36.705,Z -87.814,A -90.000,B 90.000,C 0.000} C_DIS
LIN {X -42.046,Y -36.701,Z -87.544,A -90.000,B 90.000,C 0.000} C_DIS
LIN {X -42.069,Y -36.701,Z -87.438,A -90.000,B 90.000,C 0.000} C_DIS
LIN {X -42.150,Y -36.702,Z -87.026,A -90.000,B 90.000,C 0.000} C_DIS
LIN {X -42.177,Y -36.703,Z -86.867,A -90.000,B 90.000,C 0.000} C_DIS
LIN {X -42.209,Y -36.708,Z -86.632,A -90.000,B 90.000,C 0.000} C_DIS
LIN {X -42.227,Y -36.717,Z -86.422,A -90.000,B 90.000,C 0.000} C_DIS
LIN {X -42.249,Y -36.753,Z -85.709,A -90.000,B 90.000,C 0.000} C_DIS
LIN {X -42.256,Y -36.762,Z -85.451,A -90.000,B 90.000,C 0.000} C_DIS
LIN {X -42.262,Y -36.764,Z -85.092,A -90.000,B 90.000,C 0.000} C_DIS
LIN {X -42.272,Y -36.756,Z -84.366,A -90.000,B 90.000,C 0.000} C_DIS
LIN {X -42.268,Y -36.756,Z -84.155,A -90.000,B 90.000,C 0.000} C_DIS
LIN {X -42.243,Y -36.760,Z -83.808,A -90.000,B 90.000,C 0.000} C_DIS
LIN {X -42.195,Y -36.772,Z -83.498,A -90.000,B 90.000,C 0.000} C_DIS
LIN {X -42.093,Y -36.799,Z -83.065,A -90.000,B 90.000,C 0.000} C_DIS
LIN {X -42.041,Y -36.808,Z -82.850,A -90.000,B 90.000,C 0.000} C_DIS
LIN {X -42.000,Y -36.808,Z -82.688,A -90.000,B 90.000,C 0.000} C_DIS
LIN {X -41.777,Y -36.813,Z -81.799,A -90.000,B 90.000,C 0.000} C_DIS
LIN {X -41.749,Y -36.813,Z -81.680,A -90.000,B 90.000,C 0.000} C_DIS
LIN {X -41.703,Y -36.814,Z -81.498,A -90.000,B 90.000,C 0.000} C_DIS
LIN {X -41.636,Y -36.819,Z -81.271,A -90.000,B 90.000,C 0.000} C_DIS
LIN {X -41.547,Y -36.827,Z -81.032,A -90.000,B 90.000,C 0.000} C_DIS
LIN {X -41.531,Y -36.829,Z -80.995,A -90.000,B 90.000,C 0.000} C_DIS
LIN {X -41.451,Y -36.835,Z -80.814,A -90.000,B 90.000,C 0.000} C_DIS
LIN {X -41.358,Y -36.835,Z -80.611,A -90.000,B 90.000,C 0.000} C_DIS
LIN {X -40.721,Y -36.849,Z -79.200,A -90.000,B 90.000,C 0.000} C_DIS
LIN {X -40.666,Y -36.851,Z -79.095,A -90.000,B 90.000,C 0.000} C_DIS
LIN {X -40.565,Y -36.852,Z -78.913,A -90.000,B 90.000,C 0.000} C_DIS
LIN {X -40.415,Y -36.852,Z -78.660,A -90.000,B 90.000,C 0.000} C_DIS
LIN {X -40.261,Y -36.854,Z -78.421,A -90.000,B 90.000,C 0.000} C_DIS
LIN {X -39.553,Y -36.878,Z -77.333,A -90.000,B 90.000,C 0.000} C_DIS
LIN {X -39.331,Y -36.883,Z -76.994,A -90.000,B 90.000,C 0.000} C_DIS
LIN {X -38.960,Y -36.896,Z -76.471,A -90.000,B 90.000,C 0.000} C_DIS
LIN {X -38.556,Y -36.899,Z -75.905,A -90.000,B 90.000,C 0.000} C_DIS
LIN {X -38.459,Y -36.901,Z -75.779,A -90.000,B 90.000,C 0.000} C_DIS
LIN {X -38.231,Y -36.909,Z -75.507,A -90.000,B 90.000,C 0.000} C_DIS
LIN {X -37.933,Y -36.912,Z -75.153,A -90.000,B 90.000,C 0.000} C_DIS
LIN {X -37.699,Y -36.911,Z -74.882,A -90.000,B 90.000,C 0.000} C_DIS
LIN {X -37.608,Y -36.911,Z -74.785,A -90.000,B 90.000,C 0.000} C_DIS
LIN {X -37.082,Y -36.918,Z -74.256,A -90.000,B 90.000,C 0.000} C_DIS
LIN {X -36.954,Y -36.922,Z -74.138,A -90.000,B 90.000,C 0.000} C_DIS
LIN {X -36.554,Y -36.930,Z -73.801,A -90.000,B 90.000,C 0.000} C_DIS
LIN {X -36.231,Y -36.928,Z -73.531,A -90.000,B 90.000,C 0.000} C_DIS
LIN {X -35.605,Y -36.901,Z -73.016,A -90.000,B 90.000,C 0.000} C_DIS
LIN {X -35.417,Y -36.895,Z -72.874,A -90.000,B 90.000,C 0.000} C_DIS
LIN {X -35.210,Y -36.892,Z -72.739,A -90.000,B 90.000,C 0.000} C_DIS
LIN {X -35.149,Y -36.892,Z -72.705,A -90.000,B 90.000,C 0.000} C_DIS
LIN {X -34.997,Y -36.891,Z -72.627,A -90.000,B 90.000,C 0.000} C_DIS
LIN {X -34.670,Y -36.893,Z -72.477,A -90.000,B 90.000,C 0.000} C_DIS
LIN {X -34.579,Y -36.895,Z -72.438,A -90.000,B 90.000,C 0.000} C_DIS
LIN {X -33.703,Y -36.910,Z -72.086,A -90.000,B 90.000,C 0.000} C_DIS
LIN {X -33.448,Y -36.912,Z -71.984,A -90.000,B 90.000,C 0.000} C_DIS
LIN {X -33.239,Y -36.903,Z -71.905,A -90.000,B 90.000,C 0.000} C_DIS
LIN {X -33.183,Y -36.902,Z -71.887,A -90.000,B 90.000,C 0.000} C_DIS
LIN {X -32.096,Y -36.858,Z -71.580,A -90.000,B 90.000,C 0.000} C_DIS
LIN {X -31.978,Y -36.855,Z -71.550,A -90.000,B 90.000,C 0.000} C_DIS
LIN {X -31.720,Y -36.849,Z -71.494,A -90.000,B 90.000,C 0.000} C_DIS
LIN {X -31.221,Y -36.831,Z -71.392,A -90.000,B 90.000,C 0.000} C_DIS
LIN {X -31.002,Y -36.826,Z -71.359,A -90.000,B 90.000,C 0.000} C_DIS
LIN {X -30.641,Y -36.824,Z -71.324,A -90.000,B 90.000,C 0.000} C_DIS
LIN {X -29.909,Y -36.806,Z -71.258,A -90.000,B 90.000,C 0.000} C_DIS
LIN {X -29.655,Y -36.796,Z -71.236,A -90.000,B 90.000,C 0.000} C_DIS
LIN {X -29.566,Y -36.793,Z -71.231,A -90.000,B 90.000,C 0.000} C_DIS
LIN {X -29.304,Y -36.787,Z -71.229,A -90.000,B 90.000,C 0.000} C_DIS
LIN {X -28.858,Y -36.779,Z -71.235,A -90.000,B 90.000,C 0.000} C_DIS
LIN {X -28.692,Y -36.779,Z -71.246,A -90.000,B 90.000,C 0.000} C_DIS
LIN {X -28.452,Y -36.783,Z -71.278,A -90.000,B 90.000,C 0.000} C_DIS
LIN {X -28.346,Y -36.786,Z -71.299,A -90.000,B 90.000,C 0.000} C_DIS
LIN {X -28.198,Y -36.789,Z -71.321,A -90.000,B 90.000,C 0.000} C_DIS
LIN {X -27.247,Y -36.776,Z -71.476,A -90.000,B 90.000,C 0.000} C_DIS
LIN {X -26.539,Y -36.765,Z -71.594,A -90.000,B 90.000,C 0.000} C_DIS
LIN {X -26.307,Y -36.763,Z -71.642,A -90.000,B 90.000,C 0.000} C_DIS
LIN {X -26.180,Y -36.763,Z -71.672,A -90.000,B 90.000,C 0.000} C_DIS
LIN {X -25.955,Y -36.765,Z -71.733,A -90.000,B 90.000,C 0.000} C_DIS
LIN {X -24.770,Y -36.742,Z -71.986,A -90.000,B 90.000,C 0.000} C_DIS
LIN {X -24.446,Y -36.731,Z -72.037,A -90.000,B 90.000,C 0.000} C_DIS
LIN {X -23.728,Y -36.721,Z -72.147,A -90.000,B 90.000,C 0.000} C_DIS
LIN {X -23.353,Y -36.683,Z -72.143,A -90.000,B 90.000,C 0.000} C_DIS
LIN {X -23.072,Y -36.593,Z -71.987,A -90.000,B 90.000,C 0.000} C_DIS
LIN {X -22.724,Y -36.492,Z -71.797,A -90.000,B 90.000,C 0.000} C_DIS
LIN {X -22.264,Y -36.357,Z -71.544,A -90.000,B 90.000,C 0.000} C_DIS
LIN {X -22.156,Y -36.328,Z -71.490,A -90.000,B 90.000,C 0.000} C_DIS
LIN {X -22.022,Y -36.296,Z -71.433,A -90.000,B 90.000,C 0.000} C_DIS
LIN {X -21.666,Y -36.256,Z -71.264,A -90.000,B 90.000,C 0.000} C_DIS
LIN {X -21.203,Y -36.248,Z -71.016,A -90.000,B 90.000,C 0.000} C_DIS
LIN {X -20.844,Y -36.244,Z -70.828,A -90.000,B 90.000,C 0.000} C_DIS
LIN {X -20.760,Y -36.242,Z -70.789,A -90.000,B 90.000,C 0.000} C_DIS
LIN {X -20.357,Y -36.247,Z -70.613,A -90.000,B 90.000,C 0.000} C_DIS
LIN {X -19.771,Y -36.247,Z -70.364,A -90.000,B 90.000,C 0.000} C_DIS
LIN {X -19.202,Y -36.229,Z -70.131,A -90.000,B 90.000,C 0.000} C_DIS
LIN {X -19.038,Y -36.221,Z -70.069,A -90.000,B 90.000,C 0.000} C_DIS
LIN {X -18.714,Y -36.211,Z -69.959,A -90.000,B 90.000,C 0.000} C_DIS
LIN {X -18.553,Y -36.209,Z -69.909,A -90.000,B 90.000,C 0.000} C_DIS
LIN {X -18.418,Y -36.211,Z -69.873,A -90.000,B 90.000,C 0.000} C_DIS
LIN {X -17.906,Y -36.229,Z -69.751,A -90.000,B 90.000,C 0.000} C_DIS
LIN {X -17.756,Y -36.234,Z -69.719,A -90.000,B 90.000,C 0.000} C_DIS
LIN {X -17.667,Y -36.240,Z -69.703,A -90.000,B 90.000,C 0.000} C_DIS
LIN {X -17.282,Y -36.251,Z -69.640,A -90.000,B 90.000,C 0.000} C_DIS
LIN {X -16.636,Y -36.239,Z -69.555,A -90.000,B 90.000,C 0.000} C_DIS
LIN {X -15.888,Y -36.232,Z -69.472,A -90.000,B 90.000,C 0.000} C_DIS
LIN {X -15.452,Y -36.234,Z -69.440,A -90.000,B 90.000,C 0.000} C_DIS
LIN {X -15.017,Y -36.244,Z -69.419,A -90.000,B 90.000,C 0.000} C_DIS
LIN {X -14.669,Y -36.250,Z -69.406,A -90.000,B 90.000,C 0.000} C_DIS
LIN {X -14.293,Y -36.246,Z -69.400,A -90.000,B 90.000,C 0.000} C_DIS
LIN {X -12.614,Y -36.229,Z -69.386,A -90.000,B 90.000,C 0.000} C_DIS
LIN {X -12.490,Y -36.229,Z -69.389,A -90.000,B 90.000,C 0.000} C_DIS
LIN {X -11.730,Y -36.247,Z -69.423,A -90.000,B 90.000,C 0.000} C_DIS
LIN {X -11.583,Y -36.247,Z -69.432,A -90.000,B 90.000,C 0.000} C_DIS
LIN {X -10.692,Y -36.254,Z -69.496,A -90.000,B 90.000,C 0.000} C_DIS
LIN {X -8.754,Y -36.269,Z -69.635,A -90.000,B 90.000,C 0.000} C_DIS
LIN {X -8.647,Y -36.271,Z -69.645,A -90.000,B 90.000,C 0.000} C_DIS
LIN {X -8.155,Y -36.287,Z -69.704,A -90.000,B 90.000,C 0.000} C_DIS
LIN {X -7.815,Y -36.296,Z -69.746,A -90.000,B 90.000,C 0.000} C_DIS
LIN {X -6.924,Y -36.305,Z -69.864,A -90.000,B 90.000,C 0.000} C_DIS
LIN {X -5.604,Y -36.315,Z -70.027,A -90.000,B 90.000,C 0.000} C_DIS
LIN {X -4.744,Y -36.346,Z -70.119,A -90.000,B 90.000,C 0.000} C_DIS
LIN {X -4.633,Y -36.351,Z -70.134,A -90.000,B 90.000,C 0.000} C_DIS
LIN {X -4.031,Y -36.385,Z -70.231,A -90.000,B 90.000,C 0.000} C_DIS
LIN {X -3.647,Y -36.405,Z -70.287,A -90.000,B 90.000,C 0.000} C_DIS
LIN {X -3.062,Y -36.432,Z -70.373,A -90.000,B 90.000,C 0.000} C_DIS
LIN {X -2.640,Y -36.450,Z -70.434,A -90.000,B 90.000,C 0.000} C_DIS
LIN {X -2.431,Y -36.460,Z -70.462,A -90.000,B 90.000,C 0.000} C_DIS
LIN {X -1.903,Y -36.505,Z -70.526,A -90.000,B 90.000,C 0.000} C_DIS
LIN {X -0.701,Y -36.605,Z -70.648,A -90.000,B 90.000,C 0.000} C_DIS
LIN {X 0.040,Y -36.692,Z -70.717,A -90.000,B 90.000,C 0.000} C_DIS
LIN {X 0.130,Y -36.703,Z -70.728,A -90.000,B 90.000,C 0.000} C_DIS
LIN {X 0.797,Y -36.787,Z -70.826,A -90.000,B 90.000,C 0.000} C_DIS
LIN {X 0.867,Y -36.796,Z -70.834,A -90.000,B 90.000,C 0.000} C_DIS
LIN {X 1.086,Y -36.819,Z -70.835,A -90.000,B 90.000,C 0.000} C_DIS
LIN {X 1.787,Y -36.918,Z -70.837,A -90.000,B 90.000,C 0.000} C_DIS
LIN {X 2.086,Y -36.959,Z -70.823,A -90.000,B 90.000,C 0.000} C_DIS
LIN {X 2.156,Y -36.959,Z -70.729,A -90.000,B 90.000,C 0.000} C_DIS
LIN {X 2.329,Y -36.959,Z -70.471,A -90.000,B 90.000,C 0.000} C_DIS
LIN {X 2.450,Y -36.952,Z -70.293,A -90.000,B 90.000,C 0.000} C_DIS
LIN {X 2.545,Y -36.943,Z -70.153,A -90.000,B 90.000,C 0.000} C_DIS
LIN {X 2.626,Y -36.936,Z -70.049,A -90.000,B 90.000,C 0.000} C_DIS
LIN {X 2.755,Y -36.927,Z -69.907,A -90.000,B 90.000,C 0.000} C_DIS
LIN {X 2.851,Y -36.921,Z -69.811,A -90.000,B 90.000,C 0.000} C_DIS
LIN {X 3.005,Y -36.912,Z -69.661,A -90.000,B 90.000,C 0.000} C_DIS
LIN {X 3.090,Y -36.907,Z -69.584,A -90.000,B 90.000,C 0.000} C_DIS
LIN {X 3.208,Y -36.902,Z -69.489,A -90.000,B 90.000,C 0.000} C_DIS
LIN {X 3.385,Y -36.897,Z -69.357,A -90.000,B 90.000,C 0.000} C_DIS
LIN {X 3.474,Y -36.892,Z -69.296,A -90.000,B 90.000,C 0.000} C_DIS
LIN {X 3.558,Y -36.889,Z -69.241,A -90.000,B 90.000,C 0.000} C_DIS
LIN {X 3.743,Y -36.871,Z -69.124,A -90.000,B 90.000,C 0.000} C_DIS
LIN {X 4.396,Y -36.796,Z -68.672,A -90.000,B 90.000,C 0.000} C_DIS
LIN {X 4.475,Y -36.788,Z -68.620,A -90.000,B 90.000,C 0.000} C_DIS
LIN {X 4.570,Y -36.779,Z -68.565,A -90.000,B 90.000,C 0.000} C_DIS
LIN {X 4.725,Y -36.771,Z -68.488,A -90.000,B 90.000,C 0.000} C_DIS
LIN {X 4.935,Y -36.762,Z -68.393,A -90.000,B 90.000,C 0.000} C_DIS
LIN {X 5.028,Y -36.758,Z -68.354,A -90.000,B 90.000,C 0.000} C_DIS
LIN {X 5.237,Y -36.755,Z -68.278,A -90.000,B 90.000,C 0.000} C_DIS
LIN {X 6.518,Y -36.668,Z -67.844,A -90.000,B 90.000,C 0.000} C_DIS
LIN {X 6.819,Y -36.650,Z -67.748,A -90.000,B 90.000,C 0.000} C_DIS
LIN {X 6.963,Y -36.643,Z -67.708,A -90.000,B 90.000,C 0.000} C_DIS
LIN {X 7.092,Y -36.637,Z -67.675,A -90.000,B 90.000,C 0.000} C_DIS
LIN {X 7.222,Y -36.632,Z -67.647,A -90.000,B 90.000,C 0.000} C_DIS
LIN {X 7.904,Y -36.606,Z -67.511,A -90.000,B 90.000,C 0.000} C_DIS
LIN {X 8.079,Y -36.602,Z -67.484,A -90.000,B 90.000,C 0.000} C_DIS
LIN {X 8.395,Y -36.597,Z -67.450,A -90.000,B 90.000,C 0.000} C_DIS
LIN {X 9.318,Y -36.562,Z -67.357,A -90.000,B 90.000,C 0.000} C_DIS
LIN {X 9.718,Y -36.528,Z -67.325,A -90.000,B 90.000,C 0.000} C_DIS
LIN {X 9.820,Y -36.521,Z -67.319,A -90.000,B 90.000,C 0.000} C_DIS
LIN {X 10.046,Y -36.511,Z -67.324,A -90.000,B 90.000,C 0.000} C_DIS
LIN {X 10.327,Y -36.506,Z -67.345,A -90.000,B 90.000,C 0.000} C_DIS
LIN {X 10.529,Y -36.505,Z -67.365,A -90.000,B 90.000,C 0.000} C_DIS
LIN {X 10.894,Y -36.514,Z -67.400,A -90.000,B 90.000,C 0.000} C_DIS
LIN {X 11.214,Y -36.517,Z -67.433,A -90.000,B 90.000,C 0.000} C_DIS
LIN {X 11.291,Y -36.515,Z -67.442,A -90.000,B 90.000,C 0.000} C_DIS
LIN {X 12.002,Y -36.486,Z -67.505,A -90.000,B 90.000,C 0.000} C_DIS
LIN {X 12.091,Y -36.414,Z -67.369,A -90.000,B 90.000,C 0.000} C_DIS
LIN {X 12.161,Y -36.362,Z -67.273,A -90.000,B 90.000,C 0.000} C_DIS
LIN {X 12.217,Y -36.325,Z -67.202,A -90.000,B 90.000,C 0.000} C_DIS
LIN {X 12.317,Y -36.259,Z -67.082,A -90.000,B 90.000,C 0.000} C_DIS
LIN {X 12.460,Y -36.181,Z -66.929,A -90.000,B 90.000,C 0.000} C_DIS
LIN {X 12.551,Y -36.135,Z -66.837,A -90.000,B 90.000,C 0.000} C_DIS
LIN {X 12.642,Y -36.139,Z -66.689,A -90.000,B 90.000,C 0.000} C_DIS
LIN {X 12.715,Y -36.140,Z -66.583,A -90.000,B 90.000,C 0.000} C_DIS
LIN {X 13.007,Y -36.150,Z -66.170,A -90.000,B 90.000,C 0.000} C_DIS
LIN {X 13.059,Y -36.153,Z -66.099,A -90.000,B 90.000,C 0.000} C_DIS
LIN {X 13.372,Y -36.152,Z -65.728,A -90.000,B 90.000,C 0.000} C_DIS
LIN {X 13.482,Y -36.151,Z -65.604,A -90.000,B 90.000,C 0.000} C_DIS
LIN {X 13.546,Y -36.150,Z -65.542,A -90.000,B 90.000,C 0.000} C_DIS
LIN {X 13.771,Y -36.150,Z -65.338,A -90.000,B 90.000,C 0.000} C_DIS
LIN {X 13.843,Y -36.144,Z -65.278,A -90.000,B 90.000,C 0.000} C_DIS
LIN {X 13.983,Y -36.137,Z -65.171,A -90.000,B 90.000,C 0.000} C_DIS
LIN {X 14.040,Y -36.137,Z -65.131,A -90.000,B 90.000,C 0.000} C_DIS
LIN {X 14.103,Y -36.135,Z -65.089,A -90.000,B 90.000,C 0.000} C_DIS
LIN {X 14.193,Y -36.136,Z -65.026,A -90.000,B 90.000,C 0.000} C_DIS
LIN {X 14.371,Y -36.138,Z -64.903,A -90.000,B 90.000,C 0.000} C_DIS
LIN {X 14.499,Y -36.144,Z -64.823,A -90.000,B 90.000,C 0.000} C_DIS
LIN {X 14.655,Y -36.156,Z -64.733,A -90.000,B 90.000,C 0.000} C_DIS
LIN {X 14.809,Y -36.155,Z -64.654,A -90.000,B 90.000,C 0.000} C_DIS
LIN {X 14.904,Y -36.157,Z -64.607,A -90.000,B 90.000,C 0.000} C_DIS
LIN {X 14.994,Y -36.161,Z -64.567,A -90.000,B 90.000,C 0.000} C_DIS
LIN {X 15.351,Y -36.160,Z -64.439,A -90.000,B 90.000,C 0.000} C_DIS
LIN {X 15.391,Y -36.158,Z -64.427,A -90.000,B 90.000,C 0.000} C_DIS
LIN {X 15.565,Y -36.150,Z -64.381,A -90.000,B 90.000,C 0.000} C_DIS
LIN {X 15.718,Y -36.150,Z -64.348,A -90.000,B 90.000,C 0.000} C_DIS
LIN {X 16.182,Y -36.135,Z -64.262,A -90.000,B 90.000,C 0.000} C_DIS
LIN {X 16.612,Y -36.108,Z -64.192,A -90.000,B 90.000,C 0.000} C_DIS
LIN {X 16.745,Y -36.103,Z -64.175,A -90.000,B 90.000,C 0.000} C_DIS
LIN {X 17.102,Y -36.082,Z -64.161,A -90.000,B 90.000,C 0.000} C_DIS
LIN {X 17.190,Y -36.074,Z -64.161,A -90.000,B 90.000,C 0.000} C_DIS
LIN {X 17.375,Y -36.059,Z -64.169,A -90.000,B 90.000,C 0.000} C_DIS
LIN {X 17.790,Y -36.041,Z -64.205,A -90.000,B 90.000,C 0.000} C_DIS
LIN {X 17.945,Y -36.038,Z -64.224,A -90.000,B 90.000,C 0.000} C_DIS
LIN {X 18.000,Y -36.038,Z -64.232,A -90.000,B 90.000,C 0.000} C_DIS
LIN {X 18.250,Y -36.039,Z -64.279,A -90.000,B 90.000,C 0.000} C_DIS
LIN {X 18.429,Y -36.032,Z -64.319,A -90.000,B 90.000,C 0.000} C_DIS
LIN {X 18.451,Y -36.046,Z -64.312,A -90.000,B 90.000,C 0.000} C_DIS
LIN {X 18.488,Y -36.066,Z -64.302,A -90.000,B 90.000,C 0.000} C_DIS
LIN {X 18.553,Y -36.068,Z -64.230,A -90.000,B 90.000,C 0.000} C_DIS
LIN {X 18.726,Y -36.078,Z -64.050,A -90.000,B 90.000,C 0.000} C_DIS
LIN {X 18.851,Y -36.081,Z -63.931,A -90.000,B 90.000,C 0.000} C_DIS
LIN {X 18.974,Y -36.084,Z -63.827,A -90.000,B 90.000,C 0.000} C_DIS
LIN {X 19.160,Y -36.096,Z -63.680,A -90.000,B 90.000,C 0.000} C_DIS
LIN {X 19.297,Y -36.095,Z -63.584,A -90.000,B 90.000,C 0.000} C_DIS
LIN {X 19.413,Y -36.097,Z -63.509,A -90.000,B 90.000,C 0.000} C_DIS
LIN {X 19.495,Y -36.103,Z -63.460,A -90.000,B 90.000,C 0.000} C_DIS
LIN {X 19.791,Y -36.101,Z -63.305,A -90.000,B 90.000,C 0.000} C_DIS
LIN {X 19.899,Y -36.104,Z -63.253,A -90.000,B 90.000,C 0.000} C_DIS
LIN {X 20.199,Y -36.102,Z -63.144,A -90.000,B 90.000,C 0.000} C_DIS
LIN {X 20.255,Y -36.101,Z -63.124,A -90.000,B 90.000,C 0.000} C_DIS
LIN {X 20.345,Y -36.095,Z -63.097,A -90.000,B 90.000,C 0.000} C_DIS
LIN {X 20.548,Y -36.090,Z -63.046,A -90.000,B 90.000,C 0.000} C_DIS
LIN {X 20.619,Y -36.090,Z -63.031,A -90.000,B 90.000,C 0.000} C_DIS
LIN {X 21.011,Y -36.069,Z -62.965,A -90.000,B 90.000,C 0.000} C_DIS
LIN {X 21.162,Y -36.060,Z -62.948,A -90.000,B 90.000,C 0.000} C_DIS
LIN {X 21.556,Y -36.040,Z -62.933,A -90.000,B 90.000,C 0.000} C_DIS
LIN {X 21.809,Y -36.011,Z -62.939,A -90.000,B 90.000,C 0.000} C_DIS
LIN {X 21.940,Y -36.002,Z -62.949,A -90.000,B 90.000,C 0.000} C_DIS
LIN {X 22.315,Y -35.960,Z -63.007,A -90.000,B 90.000,C 0.000} C_DIS
LIN {X 22.386,Y -35.951,Z -63.021,A -90.000,B 90.000,C 0.000} C_DIS
LIN {X 22.764,Y -35.913,Z -63.113,A -90.000,B 90.000,C 0.000} C_DIS
LIN {X 22.871,Y -35.897,Z -63.145,A -90.000,B 90.000,C 0.000} C_DIS
LIN {X 23.051,Y -35.969,Z -63.104,A -90.000,B 90.000,C 0.000} C_DIS
LIN {X 23.141,Y -36.006,Z -63.087,A -90.000,B 90.000,C 0.000} C_DIS
LIN {X 23.289,Y -36.073,Z -63.068,A -90.000,B 90.000,C 0.000} C_DIS
LIN {X 23.540,Y -36.173,Z -63.061,A -90.000,B 90.000,C 0.000} C_DIS
LIN {X 23.720,Y -36.245,Z -63.062,A -90.000,B 90.000,C 0.000} C_DIS
LIN {X 23.849,Y -36.301,Z -63.071,A -90.000,B 90.000,C 0.000} C_DIS
LIN {X 23.978,Y -36.346,Z -63.091,A -90.000,B 90.000,C 0.000} C_DIS
LIN {X 24.360,Y -36.387,Z -62.933,A -90.000,B 90.000,C 0.000} C_DIS
LIN {X 24.464,Y -36.398,Z -62.887,A -90.000,B 90.000,C 0.000} C_DIS
LIN {X 24.537,Y -36.401,Z -62.843,A -90.000,B 90.000,C 0.000} C_DIS
LIN {X 24.606,Y -36.399,Z -62.791,A -90.000,B 90.000,C 0.000} C_DIS
LIN {X 24.659,Y -36.392,Z -62.739,A -90.000,B 90.000,C 0.000} C_DIS
LIN {X 24.924,Y -36.352,Z -62.460,A -90.000,B 90.000,C 0.000} C_DIS
LIN {X 25.039,Y -36.338,Z -62.340,A -90.000,B 90.000,C 0.000} C_DIS
LIN {X 25.114,Y -36.328,Z -62.263,A -90.000,B 90.000,C 0.000} C_DIS
LIN {X 25.202,Y -36.319,Z -62.177,A -90.000,B 90.000,C 0.000} C_DIS
LIN {X 25.239,Y -36.316,Z -62.143,A -90.000,B 90.000,C 0.000} C_DIS
LIN {X 25.469,Y -36.282,Z -61.946,A -90.000,B 90.000,C 0.000} C_DIS
LIN {X 25.569,Y -36.268,Z -61.866,A -90.000,B 90.000,C 0.000} C_DIS
LIN {X 25.621,Y -36.263,Z -61.828,A -90.000,B 90.000,C 0.000} C_DIS
LIN {X 25.638,Y -36.225,Z -61.754,A -90.000,B 90.000,C 0.000} C_DIS
LIN {X 25.682,Y -36.137,Z -61.594,A -90.000,B 90.000,C 0.000} C_DIS
LIN {X 25.736,Y -36.048,Z -61.440,A -90.000,B 90.000,C 0.000} C_DIS
LIN {X 25.778,Y -35.985,Z -61.330,A -90.000,B 90.000,C 0.000} C_DIS
LIN {X 25.821,Y -35.931,Z -61.233,A -90.000,B 90.000,C 0.000} C_DIS
LIN {X 25.960,Y -35.790,Z -60.964,A -90.000,B 90.000,C 0.000} C_DIS
LIN {X 26.045,Y -35.717,Z -60.819,A -90.000,B 90.000,C 0.000} C_DIS
LIN {X 26.103,Y -35.672,Z -60.728,A -90.000,B 90.000,C 0.000} C_DIS
LIN {X 26.248,Y -35.575,Z -60.520,A -90.000,B 90.000,C 0.000} C_DIS
LIN {X 26.297,Y -35.547,Z -60.457,A -90.000,B 90.000,C 0.000} C_DIS
LIN {X 26.387,Y -35.501,Z -60.350,A -90.000,B 90.000,C 0.000} C_DIS
LIN {X 26.526,Y -35.442,Z -60.202,A -90.000,B 90.000,C 0.000} C_DIS
LIN {X 26.473,Y -35.466,Z -59.820,A -90.000,B 90.000,C 0.000} C_DIS
LIN {X 26.448,Y -35.493,Z -59.500,A -90.000,B 90.000,C 0.000} C_DIS
LIN {X 26.446,Y -35.497,Z -59.445,A -90.000,B 90.000,C 0.000} C_DIS
LIN {X 26.432,Y -35.525,Z -59.056,A -90.000,B 90.000,C 0.000} C_DIS
LIN {X 26.434,Y -35.549,Z -58.721,A -90.000,B 90.000,C 0.000} C_DIS
LIN {X 26.441,Y -35.577,Z -58.459,A -90.000,B 90.000,C 0.000} C_DIS
LIN {X 26.498,Y -35.613,Z -57.987,A -90.000,B 90.000,C 0.000} C_DIS
LIN {X 26.528,Y -35.625,Z -57.790,A -90.000,B 90.000,C 0.000} C_DIS
LIN {X 26.546,Y -35.635,Z -57.683,A -90.000,B 90.000,C 0.000} C_DIS
LIN {X 26.573,Y -35.652,Z -57.540,A -90.000,B 90.000,C 0.000} C_DIS
LIN {X 26.690,Y -35.681,Z -57.125,A -90.000,B 90.000,C 0.000} C_DIS
LIN {X 26.703,Y -35.684,Z -57.080,A -90.000,B 90.000,C 0.000} C_DIS
LIN {X 26.753,Y -35.690,Z -56.952,A -90.000,B 90.000,C 0.000} C_DIS
LIN {X 26.875,Y -35.712,Z -56.655,A -90.000,B 90.000,C 0.000} C_DIS
LIN {X 26.945,Y -35.714,Z -56.514,A -90.000,B 90.000,C 0.000} C_DIS
LIN {X 27.037,Y -35.724,Z -56.339,A -90.000,B 90.000,C 0.000} C_DIS
LIN {X 27.158,Y -35.740,Z -56.125,A -90.000,B 90.000,C 0.000} C_DIS
LIN {X 27.240,Y -35.744,Z -55.998,A -90.000,B 90.000,C 0.000} C_DIS
LIN {X 27.296,Y -35.748,Z -55.915,A -90.000,B 90.000,C 0.000} C_DIS
LIN {X 27.387,Y -35.761,Z -55.786,A -90.000,B 90.000,C 0.000} C_DIS
LIN {X 27.551,Y -35.778,Z -55.568,A -90.000,B 90.000,C 0.000} C_DIS
LIN {X 27.721,Y -35.785,Z -55.375,A -90.000,B 90.000,C 0.000} C_DIS
LIN {X 27.843,Y -35.797,Z -55.244,A -90.000,B 90.000,C 0.000} C_DIS
LIN {X 28.049,Y -35.802,Z -55.055,A -90.000,B 90.000,C 0.000} C_DIS
LIN {X 28.167,Y -35.807,Z -54.949,A -90.000,B 90.000,C 0.000} C_DIS
LIN {X 28.524,Y -35.816,Z -54.691,A -90.000,B 90.000,C 0.000} C_DIS
LIN {X 28.654,Y -35.814,Z -54.614,A -90.000,B 90.000,C 0.000} C_DIS
LIN {X 28.907,Y -35.820,Z -54.473,A -90.000,B 90.000,C 0.000} C_DIS
LIN {X 29.112,Y -35.820,Z -54.368,A -90.000,B 90.000,C 0.000} C_DIS
LIN {X 29.322,Y -35.814,Z -54.270,A -90.000,B 90.000,C 0.000} C_DIS
LIN {X 29.515,Y -35.819,Z -54.190,A -90.000,B 90.000,C 0.000} C_DIS
LIN {X 29.774,Y -35.811,Z -54.104,A -90.000,B 90.000,C 0.000} C_DIS
LIN {X 29.934,Y -35.812,Z -54.056,A -90.000,B 90.000,C 0.000} C_DIS
LIN {X 30.197,Y -35.811,Z -53.996,A -90.000,B 90.000,C 0.000} C_DIS
LIN {X 30.326,Y -35.809,Z -53.968,A -90.000,B 90.000,C 0.000} C_DIS
LIN {X 30.461,Y -35.718,Z -53.879,A -90.000,B 90.000,C 0.000} C_DIS
LIN {X 30.551,Y -35.664,Z -53.824,A -90.000,B 90.000,C 0.000} C_DIS
LIN {X 30.621,Y -35.625,Z -53.784,A -90.000,B 90.000,C 0.000} C_DIS
LIN {X 30.663,Y -35.603,Z -53.765,A -90.000,B 90.000,C 0.000} C_DIS
LIN {X 30.685,Y -35.610,Z -53.642,A -90.000,B 90.000,C 0.000} C_DIS
LIN {X 30.703,Y -35.618,Z -53.522,A -90.000,B 90.000,C 0.000} C_DIS
LIN {X 30.735,Y -35.630,Z -53.345,A -90.000,B 90.000,C 0.000} C_DIS
LIN {X 30.765,Y -35.645,Z -53.203,A -90.000,B 90.000,C 0.000} C_DIS
LIN {X 30.789,Y -35.657,Z -53.089,A -90.000,B 90.000,C 0.000} C_DIS
LIN {X 30.868,Y -35.672,Z -52.820,A -90.000,B 90.000,C 0.000} C_DIS
LIN {X 30.913,Y -35.684,Z -52.674,A -90.000,B 90.000,C 0.000} C_DIS
LIN {X 30.971,Y -35.695,Z -52.507,A -90.000,B 90.000,C 0.000} C_DIS
LIN {X 31.079,Y -35.706,Z -52.226,A -90.000,B 90.000,C 0.000} C_DIS
LIN {X 31.167,Y -35.717,Z -52.009,A -90.000,B 90.000,C 0.000} C_DIS
LIN {X 31.304,Y -35.737,Z -51.692,A -90.000,B 90.000,C 0.000} C_DIS
LIN {X 31.396,Y -35.739,Z -51.519,A -90.000,B 90.000,C 0.000} C_DIS
LIN {X 31.515,Y -35.751,Z -51.308,A -90.000,B 90.000,C 0.000} C_DIS
LIN {X 31.620,Y -35.759,Z -51.133,A -90.000,B 90.000,C 0.000} C_DIS
LIN {X 31.776,Y -35.772,Z -50.877,A -90.000,B 90.000,C 0.000} C_DIS
LIN {X 31.873,Y -35.773,Z -50.733,A -90.000,B 90.000,C 0.000} C_DIS
LIN {X 32.045,Y -35.781,Z -50.493,A -90.000,B 90.000,C 0.000} C_DIS
LIN {X 32.151,Y -35.789,Z -50.352,A -90.000,B 90.000,C 0.000} C_DIS
LIN {X 32.431,Y -35.790,Z -50.034,A -90.000,B 90.000,C 0.000} C_DIS
LIN {X 32.585,Y -35.791,Z -49.892,A -90.000,B 90.000,C 0.000} C_DIS
LIN {X 32.792,Y -35.808,Z -49.680,A -90.000,B 90.000,C 0.000} C_DIS
LIN {X 32.913,Y -35.816,Z -49.553,A -90.000,B 90.000,C 0.000} C_DIS
LIN {X 32.958,Y -35.815,Z -49.511,A -90.000,B 90.000,C 0.000} C_DIS
LIN {X 33.227,Y -35.814,Z -49.269,A -90.000,B 90.000,C 0.000} C_DIS
LIN {X 33.323,Y -35.807,Z -49.194,A -90.000,B 90.000,C 0.000} C_DIS
LIN {X 33.439,Y -35.803,Z -49.109,A -90.000,B 90.000,C 0.000} C_DIS
LIN {X 33.566,Y -35.803,Z -49.020,A -90.000,B 90.000,C 0.000} C_DIS
LIN {X 33.744,Y -35.791,Z -48.912,A -90.000,B 90.000,C 0.000} C_DIS
LIN {X 33.854,Y -35.789,Z -48.839,A -90.000,B 90.000,C 0.000} C_DIS
LIN {X 34.196,Y -35.804,Z -48.632,A -90.000,B 90.000,C 0.000} C_DIS
LIN {X 34.569,Y -35.804,Z -48.431,A -90.000,B 90.000,C 0.000} C_DIS
LIN {X 34.960,Y -35.782,Z -48.257,A -90.000,B 90.000,C 0.000} C_DIS
LIN {X 35.050,Y -35.775,Z -48.222,A -90.000,B 90.000,C 0.000} C_DIS
LIN {X 35.387,Y -35.760,Z -48.106,A -90.000,B 90.000,C 0.000} C_DIS
LIN {X 35.450,Y -35.755,Z -48.087,A -90.000,B 90.000,C 0.000} C_DIS
LIN {X 35.613,Y -35.745,Z -48.039,A -90.000,B 90.000,C 0.000} C_DIS
LIN {X 35.797,Y -35.743,Z -47.992,A -90.000,B 90.000,C 0.000} C_DIS
LIN {X 36.073,Y -35.746,Z -47.915,A -90.000,B 90.000,C 0.000} C_DIS
LIN {X 36.217,Y -35.752,Z -47.877,A -90.000,B 90.000,C 0.000} C_DIS
LIN {X 36.300,Y -35.752,Z -47.861,A -90.000,B 90.000,C 0.000} C_DIS
LIN {X 36.647,Y -35.747,Z -47.792,A -90.000,B 90.000,C 0.000} C_DIS
LIN {X 37.064,Y -35.717,Z -47.742,A -90.000,B 90.000,C 0.000} C_DIS
LIN {X 37.506,Y -35.690,Z -47.716,A -90.000,B 90.000,C 0.000} C_DIS
LIN {X 37.645,Y -35.685,Z -47.711,A -90.000,B 90.000,C 0.000} C_DIS
LIN {X 37.912,Y -35.684,Z -47.707,A -90.000,B 90.000,C 0.000} C_DIS
LIN {X 38.084,Y -35.685,Z -47.702,A -90.000,B 90.000,C 0.000} C_DIS
LIN {X 38.626,Y -35.697,Z -47.706,A -90.000,B 90.000,C 0.000} C_DIS
LIN {X 39.047,Y -35.686,Z -47.737,A -90.000,B 90.000,C 0.000} C_DIS
LIN {X 39.169,Y -35.679,Z -47.751,A -90.000,B 90.000,C 0.000} C_DIS
LIN {X 39.264,Y -35.672,Z -47.765,A -90.000,B 90.000,C 0.000} C_DIS
LIN {X 39.754,Y -35.636,Z -47.842,A -90.000,B 90.000,C 0.000} C_DIS
LIN {X 39.907,Y -35.632,Z -47.871,A -90.000,B 90.000,C 0.000} C_DIS
LIN {X 40.244,Y -35.618,Z -47.944,A -90.000,B 90.000,C 0.000} C_DIS
LIN {X 40.327,Y -35.617,Z -47.963,A -90.000,B 90.000,C 0.000} C_DIS
LIN {X 40.746,Y -35.616,Z -48.064,A -90.000,B 90.000,C 0.000} C_DIS
LIN {X 41.833,Y -35.593,Z -48.370,A -90.000,B 90.000,C 0.000} C_DIS
LIN {X 42.137,Y -35.590,Z -48.458,A -90.000,B 90.000,C 0.000} C_DIS
LIN {X 42.799,Y -35.608,Z -48.634,A -90.000,B 90.000,C 0.000} C_DIS
LIN {X 43.019,Y -35.620,Z -48.695,A -90.000,B 90.000,C 0.000} C_DIS
LIN {X 43.357,Y -35.659,Z -48.761,A -90.000,B 90.000,C 0.000} C_DIS
LIN {X 43.688,Y -35.693,Z -48.822,A -90.000,B 90.000,C 0.000} C_DIS
LIN {X 43.725,Y -35.697,Z -48.827,A -90.000,B 90.000,C 0.000} C_DIS
LIN {X 44.142,Y -35.785,Z -48.850,A -90.000,B 90.000,C 0.000} C_DIS
LIN {X 44.338,Y -35.828,Z -48.863,A -90.000,B 90.000,C 0.000} C_DIS
LIN {X 44.573,Y -35.865,Z -48.863,A -90.000,B 90.000,C 0.000} C_DIS
LIN {X 44.645,Y -35.878,Z -48.861,A -90.000,B 90.000,C 0.000} C_DIS
LIN {X 45.144,Y -35.904,Z -48.785,A -90.000,B 90.000,C 0.000} C_DIS
LIN {X 45.482,Y -35.912,Z -48.724,A -90.000,B 90.000,C 0.000} C_DIS
LIN {X 45.837,Y -35.916,Z -48.657,A -90.000,B 90.000,C 0.000} C_DIS
LIN {X 46.193,Y -35.925,Z -48.585,A -90.000,B 90.000,C 0.000} C_DIS
LIN {X 46.608,Y -35.917,Z -48.519,A -90.000,B 90.000,C 0.000} C_DIS
LIN {X 47.104,Y -35.917,Z -48.464,A -90.000,B 90.000,C 0.000} C_DIS
LIN {X 47.193,Y -35.919,Z -48.456,A -90.000,B 90.000,C 0.000} C_DIS
LIN {X 47.789,Y -35.941,Z -48.409,A -90.000,B 90.000,C 0.000} C_DIS
LIN {X 48.361,Y -35.953,Z -48.356,A -90.000,B 90.000,C 0.000} C_DIS
LIN {X 48.497,Y -35.958,Z -48.341,A -90.000,B 90.000,C 0.000} C_DIS
LIN {X 48.913,Y -35.946,Z -48.321,A -90.000,B 90.000,C 0.000} C_DIS
LIN {X 48.993,Y -35.939,Z -48.323,A -90.000,B 90.000,C 0.000} C_DIS
LIN {X 49.116,Y -35.933,Z -48.331,A -90.000,B 90.000,C 0.000} C_DIS
LIN {X 49.464,Y -35.916,Z -48.353,A -90.000,B 90.000,C 0.000} C_DIS
LIN {X 49.559,Y -35.913,Z -48.361,A -90.000,B 90.000,C 0.000} C_DIS
LIN {X 49.912,Y -35.918,Z -48.405,A -90.000,B 90.000,C 0.000} C_DIS
LIN {X 50.041,Y -35.917,Z -48.425,A -90.000,B 90.000,C 0.000} C_DIS
LIN {X 50.176,Y -35.919,Z -48.449,A -90.000,B 90.000,C 0.000} C_DIS
LIN {X 51.050,Y -35.955,Z -48.628,A -90.000,B 90.000,C 0.000} C_DIS
LIN {X 51.230,Y -35.959,Z -48.661,A -90.000,B 90.000,C 0.000} C_DIS
LIN {X 51.792,Y -35.959,Z -48.772,A -90.000,B 90.000,C 0.000} C_DIS
LIN {X 52.179,Y -35.944,Z -48.861,A -90.000,B 90.000,C 0.000} C_DIS
LIN {X 52.331,Y -35.928,Z -48.907,A -90.000,B 90.000,C 0.000} C_DIS
LIN {X 52.546,Y -35.913,Z -48.980,A -90.000,B 90.000,C 0.000} C_DIS
LIN {X 52.821,Y -35.885,Z -49.086,A -90.000,B 90.000,C 0.000} C_DIS
LIN {X 52.916,Y -35.879,Z -49.127,A -90.000,B 90.000,C 0.000} C_DIS
LIN {X 53.267,Y -35.843,Z -49.314,A -90.000,B 90.000,C 0.000} C_DIS
LIN {X 53.394,Y -35.833,Z -49.385,A -90.000,B 90.000,C 0.000} C_DIS
LIN {X 53.729,Y -35.814,Z -49.575,A -90.000,B 90.000,C 0.000} C_DIS
LIN {X 53.850,Y -35.811,Z -49.646,A -90.000,B 90.000,C 0.000} C_DIS
LIN {X 55.495,Y -35.826,Z -50.689,A -90.000,B 90.000,C 0.000} C_DIS
LIN {X 55.748,Y -35.827,Z -50.851,A -90.000,B 90.000,C 0.000} C_DIS
LIN {X 56.040,Y -35.824,Z -51.037,A -90.000,B 90.000,C 0.000} C_DIS
LIN {X 56.345,Y -35.800,Z -51.261,A -90.000,B 90.000,C 0.000} C_DIS
LIN {X 56.523,Y -35.784,Z -51.397,A -90.000,B 90.000,C 0.000} C_DIS
LIN {X 56.643,Y -35.778,Z -51.492,A -90.000,B 90.000,C 0.000} C_DIS
LIN {X 56.967,Y -35.773,Z -51.764,A -90.000,B 90.000,C 0.000} C_DIS
LIN {X 58.796,Y -35.794,Z -53.347,A -90.000,B 90.000,C 0.000} C_DIS
LIN {X 58.930,Y -35.789,Z -53.474,A -90.000,B 90.000,C 0.000} C_DIS
LIN {X 59.260,Y -35.774,Z -53.781,A -90.000,B 90.000,C 0.000} C_DIS
LIN {X 59.441,Y -35.777,Z -53.966,A -90.000,B 90.000,C 0.000} C_DIS
LIN {X 59.949,Y -35.779,Z -54.475,A -90.000,B 90.000,C 0.000} C_DIS
LIN {X 60.553,Y -35.785,Z -55.086,A -90.000,B 90.000,C 0.000} C_DIS
LIN {X 61.000,Y -35.797,Z -55.547,A -90.000,B 90.000,C 0.000} C_DIS
LIN {X 61.318,Y -35.802,Z -55.881,A -90.000,B 90.000,C 0.000} C_DIS
LIN {X 61.630,Y -35.799,Z -56.224,A -90.000,B 90.000,C 0.000} C_DIS
LIN {X 61.844,Y -35.803,Z -56.465,A -90.000,B 90.000,C 0.000} C_DIS
LIN {X 62.122,Y -35.815,Z -56.785,A -90.000,B 90.000,C 0.000} C_DIS
LIN {X 63.406,Y -35.902,Z -58.289,A -90.000,B 90.000,C 0.000} C_DIS
LIN {X 64.061,Y -35.942,Z -59.068,A -90.000,B 90.000,C 0.000} C_DIS
LIN {X 64.452,Y -35.974,Z -59.543,A -90.000,B 90.000,C 0.000} C_DIS
LIN {X 65.074,Y -36.010,Z -60.318,A -90.000,B 90.000,C 0.000} C_DIS
LIN {X 65.304,Y -36.018,Z -60.615,A -90.000,B 90.000,C 0.000} C_DIS
LIN {X 65.783,Y -36.023,Z -61.264,A -90.000,B 90.000,C 0.000} C_DIS
LIN {X 66.053,Y -36.033,Z -61.646,A -90.000,B 90.000,C 0.000} C_DIS
LIN {X 67.714,Y -36.124,Z -64.070,A -90.000,B 90.000,C 0.000} C_DIS
LIN {X 67.789,Y -36.126,Z -64.184,A -90.000,B 90.000,C 0.000} C_DIS
LIN {X 68.779,Y -36.116,Z -65.589,A -90.000,B 90.000,C 0.000} C_DIS
LIN {X 69.378,Y -36.129,Z -66.412,A -90.000,B 90.000,C 0.000} C_DIS
LIN {X 69.691,Y -36.119,Z -66.805,A -90.000,B 90.000,C 0.000} C_DIS
LIN {X 70.229,Y -36.108,Z -67.467,A -90.000,B 90.000,C 0.000} C_DIS
LIN {X 70.975,Y -36.036,Z -68.268,A -90.000,B 90.000,C 0.000} C_DIS
LIN {X 71.736,Y -36.019,Z -69.024,A -90.000,B 90.000,C 0.000} C_DIS
LIN {X 72.042,Y -36.020,Z -69.320,A -90.000,B 90.000,C 0.000} C_DIS
LIN {X 72.091,Y -36.018,Z -69.365,A -90.000,B 90.000,C 0.000} C_DIS
LIN {X 72.974,Y -35.992,Z -70.196,A -90.000,B 90.000,C 0.000} C_DIS
LIN {X 73.916,Y -35.981,Z -71.066,A -90.000,B 90.000,C 0.000} C_DIS
LIN {X 74.268,Y -35.977,Z -71.394,A -90.000,B 90.000,C 0.000} C_DIS
LIN {X 74.689,Y -35.964,Z -71.795,A -90.000,B 90.000,C 0.000} C_DIS
LIN {X 75.008,Y -35.959,Z -72.110,A -90.000,B 90.000,C 0.000} C_DIS
